DATA_BLOCK "DB_DP"   // DB85
{ S7_Optimized_Access := 'FALSE' }
// stored: AutoNumber false
   VAR RETAIN
      Anz_DP : Int := 2;   // * Anzahl Dosierpumpen
      Offset : Int := 20;   // * Beginn Daten
      leng_Pos : Int := 20;   // * Länge Daten
      DP_Nr : Int := 0;   // Nummer der aktuell bearbeiteten Pumpe
      Sekunden_Takt : Bool := FALSE;   // merkt sich den Sekundentakt
      Minuten_Takt : Bool := FALSE;   // eine Minute ist um (für einen Umlauf an)
      HandeventTakt : Bool := FALSE;   // zyklischer Abstand Meldung manuelle Zugabe
      res1 : Bool := FALSE;
      res2 : Bool := FALSE;
      res3 : Bool := FALSE;
      res4 : Bool := FALSE;
      res5 : Bool := FALSE;
      AM_Minute : Byte := 16#32;   // Altmerker Minute
      MinCount : Int := 1;   // Minutenzähler (10min)
      CheckPU : Int := 0;   // Kontrollpumpe
      resI : Int := 0;
      resD1 : DWord := 16#0000_0000;
      DP : Array[0..20] of Struct   // * Feldlänge anpassen
         Typ : Byte;   // *VAT 0=Menge Zeit,1=Menge Pulse,2=Handzugabe,5=H2O
         LaZa_Nr : Byte;   // *VAT Ladungszähler-Nr.
         EventTime : Int;   // 0=jede Dosierung sonst Zeit in Minuten
         Rest_EventTime : Int;   // Restzeit bis nächstes Event
         DP_Start : Bool;   // Start Dosierpumpe (auch extern 1 Autowert)
         DP_OFF : Bool;   // ext.Abschaltg. zB.Motorschutz oä.
         DP_Hand : Bool;   // Start eine Handzugabe
         DP_Strg : Bool;   // Störung Dosierpumpe
         DP_Imp : Bool;   // externer Zählimpuls
         DP_Niv : Bool;   // Niveau max erreicht
         DP_IN6 : Bool;
         DP_IN7 : Bool;
         DP_IN8 : Bool;
         Dosi_akt : Bool;   // Nachdosierung aktiv
         AM_Dosi : Bool;   // Altmerker Dosierung
         Meldung : Bool;   // Dosierung melden
         AM_Strg : Bool;   // Altmerker Störung
         DP_ext_Imp : Bool;   // Pumpe wird extern betrieben (Impuls wird als Eingang geliefert)
         res4 : Bool;
         AM_DP_Start : Bool;   // Merker DP Start
         RestZeit : Int;   // Restzeit Zähler Dosierimpuls/Pausenzeit
         DosMenge_Auto : Real;   // Dosiermenge Automatik
         DosMenge_Hand : Real;   // Dosiermenge Handzugabe
         ZeitBasis : Byte;   // Zeitbasis für Kalibrierung 0=s 1=min 2=h
         Korr_Einheit : Byte;   // ggf.Korrektur der Einheit
      END_STRUCT;
   END_VAR
BEGIN
   DP[0..20].Typ := 16#00;
   DP[0..20].LaZa_Nr := 16#00;
   DP[0..20].EventTime := 0;
   DP[0..7].Rest_EventTime := 1;
   DP[8..20].Rest_EventTime := 0;
   DP[0..20].DP_Start := FALSE;
   DP[0..20].DP_OFF := FALSE;
   DP[0..20].DP_Hand := FALSE;
   DP[0..20].DP_Strg := FALSE;
   DP[0..20].DP_Imp := FALSE;
   DP[0..20].DP_Niv := FALSE;
   DP[0..20].DP_IN6 := FALSE;
   DP[0..20].DP_IN7 := FALSE;
   DP[0..20].DP_IN8 := FALSE;
   DP[0..20].Dosi_akt := FALSE;
   DP[0..20].AM_Dosi := FALSE;
   DP[0..7].Meldung := TRUE;
   DP[8..20].Meldung := FALSE;
   DP[0..20].AM_Strg := FALSE;
   DP[0..20].DP_ext_Imp := FALSE;
   DP[0..20].res4 := FALSE;
   DP[0..20].AM_DP_Start := FALSE;
   DP[0..20].RestZeit := 0;
   DP[0..20].DosMenge_Auto := 0.0;
   DP[0..20].DosMenge_Hand := 0.0;
   DP[0..20].ZeitBasis := 16#00;
   DP[0..20].Korr_Einheit := 16#00;
END_DATA_BLOCK

DATA_BLOCK "DB_Dosi_Overview"   // DB88
{ S7_Optimized_Access := 'FALSE' }
// stored: AutoNumber false
   VAR RETAIN
      LZ_Count : Array[1..13] of DWord;   // * erst DZ je 1 DW
      DP_Count : Array[1..40] of DWord;   // * dann DP je 2 DW (Auto/Hand)(Feldlänge := DZ + 2*DP)
   END_VAR
BEGIN
   LZ_Count[1..13] := 16#0000_0000;
   DP_Count[1..40] := 16#0000_0000;
END_DATA_BLOCK

DATA_BLOCK "DB_NSP"   // DB96
{ S7_Optimized_Access := 'FALSE' }
// stored: AutoNumber false
   VAR RETAIN
      Anz_Per_Cyc : Int := 10;   // * Anzahl Positionen pro Zyklus (kleiner eine Sekunde müssen alle durch sein)
      Offset : Int := 20;   // Beginn Datenblock
      leng : Int := 20;   // Länge einer Struktue
      akt_NSP : Int := 55;   // aktueller Eintrag
      Test_on : Bool := TRUE;   // Testfunktion aktiv (nicht gewählte NSP/SPR aus)
      Test_akt : Bool := FALSE;   // Test Einzelpos (TestNr) aktiv
      Test_start : Bool := FALSE;   // Test angemeldet erster Umlauf alles aus
      Sekunde : Bool := FALSE;   // Sekunde M2.5 war ein
      Takt : Bool := FALSE;   // Takt (Sekunde) Zeiten zählen
      AMS_Reset : Bool := FALSE;   // Reset gefordert
      AMS_new : Bool := FALSE;   // Meldung neu schicken
      SammelWarn : Bool := FALSE;   // SammelWarnung min/max über alle Pos.
      Sammelstoer : Bool := FALSE;   // Sammelstörung Timeout über alle Pos.
      noMD_opt_max : Bool := FALSE;   // Überlauf nicht optisch melden
      noMD_opt_min : Bool := FALSE;   // Niveau min nicht optisch melden
      noMD_opt_Zeit : Bool := FALSE;   // Zeitüberschreit. nicht optisch melden
      noMD_aku_max : Bool := FALSE;   // Überlauf nicht akustisch melden
      noMD_aku_min : Bool := FALSE;   // Niveau min nicht akustisch melden
      noMD_aku_Zeit : Bool := FALSE;   // Zeitüberschreit. nicht akustisch melden
      Reset : Bool := FALSE;   // Reset Timeout NS
      TestNr : Int := 0;   // Nachspeisung für Test (alle anderen werden nicht bearbeitet)
      temp_Warn : Bool := FALSE;
      temp_STM : Bool := FALSE;
      resX122 : Bool := FALSE;
      resX123 : Bool := FALSE;
      resX124 : Bool := FALSE;
      resX125 : Bool := FALSE;
      resX126 : Bool := FALSE;
      resX127 : Bool := FALSE;
      resB1 : Byte := 16#00;
      resW1 : Int := 0;
      resD1 : DInt := 0;
      NSP : Array[1..30] of Struct
         NSP : Bool;   // Niveauregelung
         NST_in : Bool;   // Takt nach WT im Bad eingesetzt
         NST_out : Bool;   // Takt nach WT aus Bad ausgehoben
         SPR_in : Bool;   // Spritzen bei FW senkt
         SPR_out : Bool;   // Spritzen bei FW hebt
         SPR_expo : Bool;   // Spritzen während Expozeit
         SPR_Zeit : Bool;   // Spritzen feste Zeit nach Ausheben oder Einsetzen
         resTyp1 : Bool;   // ReserveTyp
         resTyp2 : Bool;   // ReserveTyp
         resTyp3 : Bool;   // ReserveTyp
         resTyp4 : Bool;   // ReserveTyp
         resTyp5 : Bool;   // ReserveTyp
         resTyp6 : Bool;   // ReserveTyp
         resTyp7 : Bool;   // ReserveTyp
         resTyp8 : Bool;   // ReserveTyp
         resTyp9 : Bool;   // ReserveTyp
         Freigabe : Bool;   // Freigabe Nachspeisung
         extern_Start : Bool;   // externe Aktivierung Taktung (zum Beispiel bei mehreren Pos)
         Niveau_ok : Bool;   // Niveau is ok Nachspeisung über Niveauregelung aus
         Nachspeisen : Bool;   // Nachspeisung aktiv --> Ventil auf / Pumpe an
         Spritzen : Bool;   // Spritzregister ein
         AL_Ueberlauf : Bool;   // Behälter Überlauf
         AL_Niv_min : Bool;   // Niveau zu niedrig --> Behälter leer
         AL_Zeit : Bool;   // Nachspeise-Zeitüberschreitung
         Restzeit_NSP : Int;   // Restzeit Nachspeisung
         TestNSP : Int;   // Testzeit Nachspeisung
         Restzeit_SPR : Int;   // Restzeit Spritzen
         VerzT : Int;   // Verzögerung Alarm Überlauf/Min-Niveau
         RestVerz : Int;   // Restzeit bis Alarm
         VerzNS_AL : Int;   // Verzögerung Alarm Nachspeisezeit zu gross
         RestNS_AL : Int;   // Restzeit bis Alarm
         AM_AL_min : Bool;   // Altmerker Alarm min
         AM_AL_Uel : Bool;   // Altmerker Alarm voll
         AM_AL_Zeit : Bool;   // Altmerker Alarm Nachspeise-Zeitüberschreitung
         AM_Bad_belegt : Bool;   // Altmerker Bad belegt
         AM_Reset : Bool;   // Altmerker RESET Nachspeise-Zeitüberschreitung
         res2 : Bool;
         res3 : Bool;
         res4 : Bool;
         SprFree : Bool;   // Spritzregister nicht bedienen (keine Ausgabe weder on noch off) Bedienung ext.
         NSPFree : Bool;   // Nachspeisung nicht bedienen (keine Ausgabe weder on noch off) Bedienung extern
         Warte_NSPT : Bool;   // getaktete Nachspeisung nicht abarbeiten
         res8 : Bool;
         res9 : Bool;
         res10 : Bool;
         res11 : Bool;
         res12 : Bool;
      END_STRUCT;
   END_VAR
BEGIN
   NSP[1..30].NSP := FALSE;
   NSP[1..30].NST_in := FALSE;
   NSP[1..30].NST_out := FALSE;
   NSP[1..30].SPR_in := FALSE;
   NSP[1..25].SPR_out := FALSE;
   NSP[26].SPR_out := TRUE;
   NSP[27..29].SPR_out := FALSE;
   NSP[30].SPR_out := TRUE;
   NSP[1..30].SPR_expo := FALSE;
   NSP[1..30].SPR_Zeit := FALSE;
   NSP[1..30].resTyp1 := FALSE;
   NSP[1..30].resTyp2 := FALSE;
   NSP[1..30].resTyp3 := FALSE;
   NSP[1..30].resTyp4 := FALSE;
   NSP[1..30].resTyp5 := FALSE;
   NSP[1..30].resTyp6 := FALSE;
   NSP[1..30].resTyp7 := FALSE;
   NSP[1..30].resTyp8 := FALSE;
   NSP[1..30].resTyp9 := FALSE;
   NSP[1..30].Freigabe := FALSE;
   NSP[1..30].extern_Start := FALSE;
   NSP[1..30].Niveau_ok := FALSE;
   NSP[1..30].Nachspeisen := FALSE;
   NSP[1..30].Spritzen := FALSE;
   NSP[1..30].AL_Ueberlauf := FALSE;
   NSP[1..30].AL_Niv_min := FALSE;
   NSP[1..30].AL_Zeit := FALSE;
   NSP[1..30].Restzeit_NSP := 0;
   NSP[1..30].TestNSP := 0;
   NSP[1..30].Restzeit_SPR := 0;
   NSP[1..30].VerzT := 0;
   NSP[1..30].RestVerz := 0;
   NSP[1..30].VerzNS_AL := 0;
   NSP[1..30].RestNS_AL := 0;
   NSP[1..30].AM_AL_min := FALSE;
   NSP[1..30].AM_AL_Uel := FALSE;
   NSP[1..30].AM_AL_Zeit := FALSE;
   NSP[1..30].AM_Bad_belegt := FALSE;
   NSP[1..30].AM_Reset := FALSE;
   NSP[1..30].res2 := FALSE;
   NSP[1..30].res3 := FALSE;
   NSP[1..30].res4 := FALSE;
   NSP[1..30].SprFree := FALSE;
   NSP[1..30].NSPFree := FALSE;
   NSP[1..30].Warte_NSPT := FALSE;
   NSP[1..30].res8 := FALSE;
   NSP[1..30].res9 := FALSE;
   NSP[1..30].res10 := FALSE;
   NSP[1..30].res11 := FALSE;
   NSP[1..30].res12 := FALSE;
END_DATA_BLOCK

DATA_BLOCK "DB_Panel_DP"   // DB86
{ S7_Optimized_Access := 'FALSE' }
AUTHOR : KHE_RE
NAME : DB_LADUN
VERSION : 2.0
// stored: AutoNumber false
   VAR RETAIN
      Anz_DP : Int := 8;   // * Anzahl Dosierpumpen
      Offset : Int := 20;   // * Beginn Daten
      Length : Int := 40;   // * Länge Daten
      res60 : Bool := FALSE;
      resB7 : Byte := 16#00;
      resB8 : Byte := 16#00;
      resB9 : Byte := 16#00;
      resB10 : Byte := 16#00;
      resB11 : Byte := 16#00;
      resD12 : DWord := 16#0000_0000;
      resD16 : DWord := 16#0000_0000;
      DoPu : Array[1..20] of Struct   // * Feldlänge anpassen
         Impulsdauer : Int;   // * Laufzeit Dosierimpuls [1/10 sec] (Falls keine Einstellmöglichkeit am PC)
         Impulspause : Int;   // * Pausenzeit zwischen zwei Impulsen [1/10 sec](Falls keine Einstellmöglichkeit
         resI : Int;
         Ein : Bool;   // Pumpe dauerhaft ein
         Auto : Bool;   // Pumpe Automatikbetrieb ein
         Kalibrierung : Bool;   // Pumpe in Kalibrierung
         res1 : Bool;
         res2 : Bool;
         Hand : Bool;   // Handdosierung läuft
         ON : Bool;   // DuPu läuft
         STM : Bool;   // DoPu Störung
         Kali_Start : Bool;   // Kalibrierung starten
         Kali_Stop : Bool;   // Kalibrierung anhalten
         res8 : Bool;
         res9 : Bool;
         res10 : Bool;
         res11 : Bool;
         res12 : Bool;
         res13 : Bool;
         Pumpleistung : Real;   // ml/s ml/Imp ....
         Zugabe_Hand : Real;   // ml
         Zugabe_Auto : Real;   // ml, ml/dm2
         RestDosierWert : Real;   // ml, Liter, g, kg usw.
         Kalibrierwert : Real;
         resD1 : DWord;
         resD2 : DWord;
         Kali_Count : DInt;   // Zählzelle Kalibrierdauer
      END_STRUCT;
   END_VAR
BEGIN
   DoPu[1..20].Impulsdauer := 1;
   DoPu[1..20].Impulspause := 1;
   DoPu[1..20].resI := 1;
   DoPu[1..20].Ein := FALSE;
   DoPu[1..4].Auto := TRUE;
   DoPu[5..20].Auto := FALSE;
   DoPu[1..20].Kalibrierung := FALSE;
   DoPu[1..20].res1 := FALSE;
   DoPu[1..20].res2 := FALSE;
   DoPu[1..20].Hand := FALSE;
   DoPu[1..20].ON := FALSE;
   DoPu[1..20].STM := FALSE;
   DoPu[1..20].Kali_Start := FALSE;
   DoPu[1..20].Kali_Stop := FALSE;
   DoPu[1..20].res8 := FALSE;
   DoPu[1..20].res9 := FALSE;
   DoPu[1..20].res10 := FALSE;
   DoPu[1..20].res11 := FALSE;
   DoPu[1..20].res12 := FALSE;
   DoPu[1..20].res13 := FALSE;
   DoPu[1..8].Pumpleistung := 0.1;
   DoPu[9..20].Pumpleistung := 0.0;
   DoPu[1..20].Zugabe_Hand := 0.0;
   DoPu[1..4].Zugabe_Auto := 10.0;
   DoPu[5..20].Zugabe_Auto := 0.0;
   DoPu[1].RestDosierWert := 0.0;
   DoPu[2].RestDosierWert := 0.09993901;
   DoPu[3..4].RestDosierWert := 0.09999623;
   DoPu[5..20].RestDosierWert := 0.0;
   DoPu[1..20].Kalibrierwert := 0.0;
   DoPu[1..20].resD1 := 16#0000_0000;
   DoPu[1..20].resD2 := 16#0000_0000;
   DoPu[1..20].Kali_Count := 0;
END_DATA_BLOCK

DATA_BLOCK "DB_Panel_LZ"   // DB81
{ S7_Optimized_Access := 'FALSE' }
AUTHOR : KHE_RE
NAME : DB_LADUN
VERSION : 2.0
// stored: AutoNumber false
   VAR RETAIN
      Anz : Int := 0;   // wird aus DB1 übernommen
      Offset : Int := 20;   // * Beginn Daten
      Length : Int := 36;   // * Länge Daten
      resB6 : Byte := 16#00;
      resB7 : Byte := 16#00;
      resD8 : DWord := 16#0000_0000;
      resD12 : DWord := 16#0000_0000;
      resD16 : DWord := 16#0000_0000;
      Becken : Array[1..20] of Struct   // * Feldlänge anpassen
         Dosi_Int : DInt;   // Abstand zw. 2 Dosierungen (Sollw.)
         Dosi_Zaehl : DInt;   // Ladung nach letzter Dosierung (Istw.)
         Rest_Zaehl1 : DInt;
         Ladu_Zaehl1 : DInt;   // kont. Ladungszähler 1 (Soll/Istw.)
         Ladu_Zaehl2 : DInt;   // kont. Ladungszähler 2 (Soll/Istw.)
         Ladu_Zaehl3 : DInt;   // kont. Ladungszähler 3 (Soll/Istw.)
         Ladu_Zaehl4 : DInt;   // kont. Ladungszähler 4 (Soll/Istw.)
         Ladu_Zaehl5 : DInt;   // kont. Ladungszähler 5 (Soll/Istw.)
         Ladu_Zaehl6 : DInt;   // kont. Ladungszähler 6 (Soll/Istw.)
      END_STRUCT;
   END_VAR
BEGIN
   Becken[1..20].Dosi_Int := 1000;
   Becken[1..20].Dosi_Zaehl := 0;
   Becken[1..20].Rest_Zaehl1 := 0;
   Becken[1..20].Ladu_Zaehl1 := 0;
   Becken[1..20].Ladu_Zaehl2 := 0;
   Becken[1..20].Ladu_Zaehl3 := 0;
   Becken[1..20].Ladu_Zaehl4 := 0;
   Becken[1..20].Ladu_Zaehl5 := 0;
   Becken[1..20].Ladu_Zaehl6 := 0;
END_DATA_BLOCK

DATA_BLOCK "DB_Panel_OVERVIEW"   // DB50
{ S7_Optimized_Access := 'FALSE' }
// stored: AutoNumber false
   VAR
      BA : Struct
         Not_Aus : Bool := FALSE;   // Not-Aus ist betätigt
         free0 : Bool := FALSE;   // sonst Anlage vom PC bedienen, nur bei BA-Schalter auf Auto
         free1 : Bool := FALSE;   // sonst Automatikbetrieb ist nicht freigegeben
         Tippbetrieb : Bool := FALSE;   // Tippbetrieb
         Handbetrieb : Bool := TRUE;   // Handbetrieb
         Automat_ein : Bool := FALSE;   // Automatikbetrieb möglich
         Automat_aus : Bool := FALSE;   // Automatikbetrieb nicht möglich
         Anlauf_Auto : Bool := FALSE;   // Anlauf Automatik für Scanvorgang WT-Positionen auf letzte Automatikposition
         Einfahr_Stop : Bool := FALSE;   // Stoppt die Einfahrt von WT in die Anlage(Feierabendprogramm)
         Mess_on : Bool := FALSE;   // Einmessung aktiv
         Taktwechsel : Bool := FALSE;   // Taktwechsel durchführen
         SIM_HISPEED : Bool := FALSE;   // Simulation erfolgt mit doppelter Geschwindigkeit
         Simulation : Bool := TRUE;   // Simulation eingeschaltet
         COM_RST : Bool := TRUE;   // Complete Restart
         FP_Automat_ein : Bool := FALSE;   // Flankenmerker positive Flanke Taste Automat ein
         newConfig : Bool := FALSE;   // neue Konfiguration (Daten neu verteilen)
      END_STRUCT;
      Offset : Int := 50;
      Leng : Int := 40;
      resW : Word := 16#0000;
      resDW2 : DWord := 16#0000_0000;
      resDW3 : DWord := 16#0000_0000;
      last_Takt : DInt := 0;
      Taktzeit : DInt := 0;   // Zeit die der Takt läuft
      Takt_Ware : DInt := 0;   // Zeit seit Ausfahrt letzte Fertigware
      resW1 : Word := 16#0000;
      Stop_Anlage : Byte := 16#00;   // ungleich 0-->Kettenbearbeitung anhalten
      Feierabend : Byte := 16#00;   // ungleich 0-->FEIERABENDPROGRAMM
      Sonder_BA : Byte := 16#00;   // ungleich 0-->ELEKTROLYSE, ENTMETALLISIEREN
      IST_Sonder_BA : Byte := 16#00;
      FB_FW_akt : Word := 16#0000;   // an Fernbedienung gewählter FW
      SPS_getaktet : Bool := TRUE;
      resDW9 : Word := 16#0000;
      Systime : DInt := 0;
      WT_Frueh : Byte := 16#00;   // Anzeige Anzahl der fertiggestellten WTs in der Frühschicht
      WT_Spaet : Byte := 16#15;   // Anzeige Anzahl der fertiggestellten WTs in der Spätschicht
      WT_Nacht : Byte := 16#00;   // Anzeige Anzahl der fertiggestellten WTs in der Nachtschicht
      resB : Byte := 16#00;
      resI : Int := 0;
      Pos : Array[1..30] of Struct   // * Feldlänge anpassen
         WT_Nr_lang : DInt;   // Warenträger-Nr lang
         WT_Nr_kurz : Byte;   // Warenträger-Nr kurz DB
         Stange_Nr : Byte;   // Warenstangen-Nr. (falls vorhanden)
         Soll_Expo : DInt;   // Sollwert Expositionszeit
         Rest_Expo : DInt;   // Verbleibende Expositionszeit
         BE_rdy : Bool;   // Beladestand bereit
         BE_leer : Bool;   // Beladestand leer
         BE_WT_vorhanden : Bool;   // Beladestand mit nicht aufgebbaren WT belegt
         BE_verriegelt : Bool;   // Beladestand angedockt und verriegelt(arretiert)
         BE_gelb : Bool;
         BE_rot : Bool;
         BE_Charge_ok : Bool;   // Behandlung fehlerfrei
         BE_Charge_nok : Bool;   // Fehler bei Behandlung
         Sonderfkt : Byte;   // Sonderfunktionen frei verwendbar(WT-Kennung)
         priorisiert : Bool;   // priorisierter WT im Bad
         in_Anlage : Bool;   // will in die Anlage
         in_Entm : Bool;   // will in die Entmetallisierung
         aus_Anlage : Bool;   // kommt aus der Anlage
         aus_Entm : Bool;   // kommt aus der Entmetallisierung
         Speicher : Bool;   // Speicherprogramm
         Warnung : Bool;   // in Position wurde eine Warnung ausgelöst
         Alarm : Bool;   // in position wurde ein Alarm ausgelöst
         belegt : Bool;   // Bad belegt
         Trommel : Bool;   // Trommelware im Bad
         Leer_WT : Bool;   // Leerstange im Bad
         Vorruf : Bool;   // Vorruf für Fahrwagen ausgelößt
         fertig : Bool;   // Expozeit abgelaufen WT zu Abholung bereit
         Sperre_in : Bool;   // Einfahrsperre
         Sperre_FW : Bool;   // Überfahrsperre
         Sperre_out : Bool;   // Ausfahrsperre
         Befx : Int;   // Befehlsindex
         Vorsperre : Bool;   // Einfahrsperre angemeldet
         Dummy1 : Bool;   // Dummy auf Dummyposition abgelegt
         Dummy2 : Bool;   // Dummy auf Mittenposition abgelegt
         Dkl_auf_Pos : Bool;   // Deckel auf dieser Position
         Expo_Warn : Bool;   // Warnung: Toleranzüberschreitg.Expozeit
         Expo_Off : Bool;   // Expositionszeit eingefroren
         NSP_ON : Bool;   // Laufanzeige Nachspeisung
         SPR_ON : Bool;   // Laufanzeige Spritzregister
         WT_Typ : Byte;   // Art des Warenträgers (z.Bsp. bei fester Zuordnung Ware-WT)
         Verweilzeit : DInt;   // Verweilzeit in s
         Sonderwert_1 : Real;   // z.B. Gewicht bei Beladestand
         Fertigzeitpunkt : DInt;   // Systemzeit PC, wann WT voraussichtlich fertig
         Sonderwert_2 : Real;   // z.B. Gewicht bei Beladestand
         resb : Byte;
         Dkl_zu : Bool;   // Deckel ist zu
         Dkl_auf : Bool;   // Deckel ist auf
         res392 : Bool;
         res393 : Bool;
         PendelHub : Bool;   // Mehrfachtauchen
         res395 : Bool;
         res396 : Bool;
         res397 : Bool;
      END_STRUCT;
   END_VAR
BEGIN
   Pos[1..30].WT_Nr_lang := 0;
   Pos[1..30].WT_Nr_kurz := 16#00;
   Pos[1..30].Stange_Nr := 16#00;
   Pos[1].Soll_Expo := 0;
   Pos[2].Soll_Expo := 360;
   Pos[3].Soll_Expo := 60;
   Pos[4..7].Soll_Expo := 1260;
   Pos[8..9].Soll_Expo := 90;
   Pos[10].Soll_Expo := 75;
   Pos[11..12].Soll_Expo := 5;
   Pos[13..14].Soll_Expo := 75;
   Pos[15..16].Soll_Expo := 5;
   Pos[17].Soll_Expo := 75;
   Pos[18].Soll_Expo := 5;
   Pos[19].Soll_Expo := 75;
   Pos[20].Soll_Expo := 5;
   Pos[21].Soll_Expo := 10;
   Pos[22].Soll_Expo := 360;
   Pos[23..27].Soll_Expo := 5;
   Pos[28].Soll_Expo := 0;
   Pos[29..30].Soll_Expo := 5;
   Pos[1..30].Rest_Expo := 0;
   Pos[1].BE_rdy := TRUE;
   Pos[2..30].BE_rdy := FALSE;
   Pos[1..30].BE_leer := FALSE;
   Pos[1..30].BE_WT_vorhanden := FALSE;
   Pos[1].BE_verriegelt := TRUE;
   Pos[2..30].BE_verriegelt := FALSE;
   Pos[1..30].BE_gelb := FALSE;
   Pos[1..30].BE_rot := FALSE;
   Pos[1..30].BE_Charge_ok := FALSE;
   Pos[1..30].BE_Charge_nok := FALSE;
   Pos[1..30].Sonderfkt := 16#00;
   Pos[1..30].priorisiert := FALSE;
   Pos[1..30].in_Anlage := FALSE;
   Pos[1..30].in_Entm := FALSE;
   Pos[1..30].aus_Anlage := FALSE;
   Pos[1..30].aus_Entm := FALSE;
   Pos[1..30].Speicher := FALSE;
   Pos[1..30].Warnung := FALSE;
   Pos[1..30].Alarm := FALSE;
   Pos[1..30].belegt := FALSE;
   Pos[1..30].Trommel := FALSE;
   Pos[1..30].Leer_WT := FALSE;
   Pos[1..30].Vorruf := FALSE;
   Pos[1..30].fertig := FALSE;
   Pos[1..30].Sperre_in := FALSE;
   Pos[1..30].Sperre_FW := FALSE;
   Pos[1..30].Sperre_out := FALSE;
   Pos[1..30].Befx := 0;
   Pos[1..30].Vorsperre := FALSE;
   Pos[1..30].Dummy1 := FALSE;
   Pos[1..30].Dummy2 := FALSE;
   Pos[1..30].Dkl_auf_Pos := FALSE;
   Pos[1..30].Expo_Warn := FALSE;
   Pos[1..30].Expo_Off := FALSE;
   Pos[1..30].NSP_ON := FALSE;
   Pos[1..30].SPR_ON := FALSE;
   Pos[1..30].WT_Typ := 16#00;
   Pos[1..30].Sonderwert_1 := 0.0;
   Pos[1..30].Fertigzeitpunkt := 0;
   Pos[1..30].Sonderwert_2 := 0.0;
   Pos[1..30].resb := 16#00;
   Pos[1..30].Dkl_zu := FALSE;
   Pos[1..30].Dkl_auf := FALSE;
   Pos[1..30].res392 := FALSE;
   Pos[1..30].res393 := FALSE;
   Pos[1..30].PendelHub := FALSE;
   Pos[1..30].res395 := FALSE;
   Pos[1..30].res396 := FALSE;
   Pos[1..30].res397 := FALSE;
END_DATA_BLOCK

DATA_BLOCK "DB_Zaehler"   // DB80
{ S7_Optimized_Access := 'FALSE' }
AUTHOR : KHE_RE
NAME : DB_LADUN
VERSION : 2.0
// stored: AutoNumber false
   VAR RETAIN
      Anz_Beck : Int := 2;   // wird aus DB1 übernommen
      Offset : Int := 40;   // * Beginn Daten
      leng_Pos : Int := 40;   // * Länge Daten
      Tag_neu : Bool := FALSE;
      Wo_neu : Bool := FALSE;
      Mo_neu : Bool := FALSE;
      res3 : Bool := FALSE;
      res4 : Bool := FALSE;
      res5 : Bool := FALSE;
      res6 : Bool := FALSE;
      AM_Takt : Bool := FALSE;
      I_Time : Byte := 16#01;
      Beck_Nr : Byte := 16#02;
      resb0 : Byte := 16#00;
      MZ_T : Byte := 16#10;   // Merkzelle akt.Tag
      MZ_W : Byte := 16#00;   // Merkzelle akt.Woche
      MZ_M : Byte := 16#06;   // Merkzelle akt.Monat
      Beck_ext : Byte := 16#00;   // Becken-Nr. für externe Dosierzähler
      Wert_Ext : Real := 0.0;   // ext. Zählwert (siehe FC6)
      resDW2 : DWord := 16#0000_0000;
      resDW3 : DWord := 16#0000_0000;
      resDW4 : DWord := 16#0000_0000;
      DosMenge_Typ7 : DWord := 16#0000_0000;
      resDW5 : DWord := 16#0000_0000;
      resW : Word := 16#0000;
      Becken : Array[1..20] of Struct   // * Feldlänge anpassen
         Typ : Byte;   // Typ 0=Ah, 1=Amin, 4=dm2, 6=ext.Zähler(FC6) 8=ext.Ah-Zähler
         Anz_Bad : Byte;   // Anz. des Bäder im Becken
         Input : Array[1..10] of Struct   // Liste der Bäder
            Pos : Int;
         END_STRUCT;
         Zaehl_int : Real;   // interner Restzähler
         Dig_Inp : Byte;   // Dig. Eing. (res.)
         Event : Bool;   // Event Mengenlimit erreicht
         Stop : Bool;   // Dosierzähler gestoppt (von DoPu o.ä.)
         res2 : Bool;
         res3 : Bool;
         res4 : Bool;
         res5 : Bool;
         res6 : Bool;
         Anf_Stp : Bool;   // kumulat.Anforderung Stop DoZa
         resW : Word;
         EventCount : Real;   // Zählzelle für Events
         ext_Val : Real;   // externer Zählwert
         AM_belegt : Word;   // Altmerker Pos.belegt
      END_STRUCT;
   END_VAR
BEGIN
   Becken[1..2].Typ := 16#05;
   Becken[3..20].Typ := 16#00;
   Becken[1..2].Anz_Bad := 16#06;
   Becken[3..20].Anz_Bad := 16#00;
   Becken[1].Input[1].Pos := 1;
   Becken[1].Input[2].Pos := 2;
   Becken[1].Input[3].Pos := 3;
   Becken[1].Input[4].Pos := 4;
   Becken[1].Input[5].Pos := 5;
   Becken[1].Input[6].Pos := 6;
   Becken[1].Input[7..10].Pos := 0;
   Becken[2].Input[1].Pos := 13;
   Becken[2].Input[2].Pos := 14;
   Becken[2].Input[3].Pos := 15;
   Becken[2].Input[4].Pos := 16;
   Becken[2].Input[5].Pos := 17;
   Becken[2].Input[6].Pos := 18;
   Becken[2].Input[7..10].Pos := 0;
   Becken[3].Input[1..10].Pos := 0;
   Becken[4].Input[1..10].Pos := 0;
   Becken[5].Input[1..10].Pos := 0;
   Becken[6].Input[1..10].Pos := 0;
   Becken[7].Input[1..10].Pos := 0;
   Becken[8].Input[1..10].Pos := 0;
   Becken[9].Input[1..10].Pos := 0;
   Becken[10].Input[1..10].Pos := 0;
   Becken[11].Input[1..10].Pos := 0;
   Becken[12].Input[1..10].Pos := 0;
   Becken[13].Input[1..10].Pos := 0;
   Becken[14].Input[1..10].Pos := 0;
   Becken[15].Input[1..10].Pos := 0;
   Becken[16].Input[1..10].Pos := 0;
   Becken[17].Input[1..10].Pos := 0;
   Becken[18].Input[1..10].Pos := 0;
   Becken[19].Input[1..10].Pos := 0;
   Becken[20].Input[1..10].Pos := 0;
   Becken[1..20].Zaehl_int := 0.0;
   Becken[1..20].Dig_Inp := 16#00;
   Becken[1..20].Event := FALSE;
   Becken[1..20].Stop := FALSE;
   Becken[1..20].res2 := FALSE;
   Becken[1..20].res3 := FALSE;
   Becken[1..20].res4 := FALSE;
   Becken[1..20].res5 := FALSE;
   Becken[1..20].res6 := FALSE;
   Becken[1..20].Anf_Stp := FALSE;
   Becken[1..20].resW := 16#0000;
   Becken[1..20].EventCount := 0.0;
   Becken[1..20].ext_Val := 0.0;
   Becken[1..20].AM_belegt := 16#0000;
END_DATA_BLOCK

DATA_BLOCK "DB_BE_Stand"   // DB4
{ S7_Optimized_Access := 'FALSE' }
// stored: AutoNumber false
   VAR RETAIN
      Anzahl : Int := 6;   // * Anzahl der BE-/Entladestände
      leng : Int := 12;   // * Länge einer Struktur
      Offset : Int := 10;   // * Beginn des Datenfeldes
      Next : Byte := 16#00;   // nächster Wt für die Anlage
      Entm : Byte := 16#00;   // nächster Wt für die Entmetallisierung
      AnfQ : Byte := 16#00;   // Anforderung Quelle
      AnfZ : Byte := 16#00;   // Anforderung Ziel
      Stand : Array[1..6] of Struct   // * Feldlänge anpassen
         Pos_Nr : USInt;
         Aufgabe_erlaubt : Bool;   // Aufgabe ist möglich
         kein_WT : Bool;   // Stand ist leer (WT ist weder physikalisch noch logisch vorhanden)
         WT_aufgegeben : Bool;   // Warenträger ist aufgegeben
         verriegelt : Bool;   // Bedienung durch FW möglich
         gelb : Bool;
         rot : Bool;
         Charge_ok : Bool;   // Behandlung war fehlerfrei
         Charge_nok : Bool;   // Behandlung war gestört
         IN_innen : Bool;   // Wagen angedockt
         IN_aussen : Bool;   // Wagen im Beladebereich
         IN_Belegt : Bool;   // WT auf Wagen
         IN_Freigabe : Bool;   // Freigabetaste (wennvorhanden über Flankenmerker Bit4.0)
         OUT_Sperre_in : Bool;   // Einfahrsperre
         OUT_Sperre_FW : Bool;   // Überfahrsperre
         OUT_Sperre_out : Bool;   // Ausfahrsperre
         OUT_FW_kommt : Bool;   // Meldung FW kommt
         Del_Count : Byte;   // Sekundenzähler zum löschen der WT-Info
         AM_Freigabe : Bool;   // Altmerker Freigabetaste
         AM_Wagen : Bool;   // Altmerker Wagen vorhanden
         res3 : Bool;
         Trommel_BE : Bool;   // Trommelstand
         Gestell_BE : Bool;   // Gestellstand
         Ausf_Ware : Bool;   // Ausfahrt Ware erlaubt
         Ausf_Entm : Bool;   // Ausfahrt entmetallisierte Gestelle
         last_WT_Trommel : Bool;   // letzter WT war / ist Trommel
         Anf_Pos : Byte;   // Position die BE-Anfordert
         last_WT : DInt;   // letzte WT-Nr-lang
         Del_All : Bool;   // 0=Programm löschen 1=gesamten WT löschen
         Auto_Delete : Bool;   // automatisches löschen fertiger WT
         Afg_WT_Nr : Bool;   // Aufgabe auch bei WT_Nr_lang<>0 erlaubt
         res1 : Bool;
         res2 : Bool;
         res4 : Bool;
         res5 : Bool;
         schnell : Bool;
         resB : Byte;
      END_STRUCT;
      Langware_vorn : Bool;
      Langware_hinten : Bool;
   END_VAR
BEGIN
   Stand[1].Pos_Nr := 25;
   Stand[2].Pos_Nr := 26;
   Stand[3].Pos_Nr := 27;
   Stand[4].Pos_Nr := 28;
   Stand[5].Pos_Nr := 29;
   Stand[6].Pos_Nr := 30;
   Stand[1..5].Aufgabe_erlaubt := FALSE;
   Stand[1..3].kein_WT := TRUE;
   Stand[4..5].kein_WT := FALSE;
   Stand[1..5].WT_aufgegeben := FALSE;
   Stand[1].verriegelt := FALSE;
   Stand[2].verriegelt := TRUE;
   Stand[3..5].verriegelt := FALSE;
   Stand[1..5].gelb := FALSE;
   Stand[1..5].rot := FALSE;
   Stand[1..5].Charge_ok := FALSE;
   Stand[1..5].Charge_nok := FALSE;
   Stand[1].IN_innen := FALSE;
   Stand[2].IN_innen := TRUE;
   Stand[3..5].IN_innen := FALSE;
   Stand[1].IN_aussen := FALSE;
   Stand[2].IN_aussen := TRUE;
   Stand[3..5].IN_aussen := FALSE;
   Stand[1..5].IN_Belegt := FALSE;
   Stand[1].IN_Freigabe := FALSE;
   Stand[2].IN_Freigabe := TRUE;
   Stand[3..5].IN_Freigabe := FALSE;
   Stand[1].OUT_Sperre_in := TRUE;
   Stand[2..5].OUT_Sperre_in := FALSE;
   Stand[1..5].OUT_Sperre_FW := FALSE;
   Stand[1..2].OUT_Sperre_out := TRUE;
   Stand[3..5].OUT_Sperre_out := FALSE;
   Stand[1..5].OUT_FW_kommt := FALSE;
   Stand[1].Del_Count := 16#05;
   Stand[2].Del_Count := 16#1E;
   Stand[3..5].Del_Count := 16#00;
   Stand[1..5].AM_Freigabe := FALSE;
   Stand[1..2].AM_Wagen := TRUE;
   Stand[3..5].AM_Wagen := FALSE;
   Stand[1..5].res3 := FALSE;
   Stand[1..5].Trommel_BE := FALSE;
   Stand[1..5].Gestell_BE := FALSE;
   Stand[1..5].Ausf_Ware := FALSE;
   Stand[1..5].Ausf_Entm := FALSE;
   Stand[1..5].last_WT_Trommel := FALSE;
   Stand[1..5].Anf_Pos := 16#00;
   Stand[1..5].last_WT := 0;
   Stand[1..2].Del_All := TRUE;
   Stand[3..5].Del_All := FALSE;
   Stand[1].Auto_Delete := FALSE;
   Stand[2].Auto_Delete := TRUE;
   Stand[3..5].Auto_Delete := FALSE;
   Stand[1..5].Afg_WT_Nr := FALSE;
   Stand[1..5].res1 := FALSE;
   Stand[1..5].res2 := FALSE;
   Stand[1..5].res4 := FALSE;
   Stand[1..5].res5 := FALSE;
   Stand[1..5].schnell := FALSE;
   Stand[1..5].resB := 16#00;
END_DATA_BLOCK

DATA_BLOCK "DB_Prog_edit"   // DB800
{ S7_Optimized_Access := 'FALSE' }
// stored: AutoNumber false
   VAR RETAIN
      akt_edit_prog : Int;
      akt_Aufgabe_Prog : Int;
      old_Aufgabe_Prog : Int;   // Hilfsvariable um Programm in Aufgabestruktur zu kopieren
      resW : Int;
      resW_1 : Int;
      resD : DInt;
      Variante : USInt;   // 1=KSvl, 2=KSvr, 3=GOli, 4= GOre,5=KShl, 6=kshr, 7=LSv(BE1), 8= LSh(BE5)
      StandNr : USInt;
      GZ_Charge : DInt;
      Prog : Array[1..100] of Struct
         "Name" : String[100];
         Geometrie : USInt;   // 0=k.A., 1=KS, 2=LS, 3=GO
         ParaByte : USInt;   // .0=lgsm senken, .1=lgsm heben
         Faktor_ATZ : Real;
         resD : DInt;
         resW : Int;
         CM03_VorSpuel : Struct
            Expo : Time_Of_Day;
            Anfahren : Bool;
            res : Bool;
            res_1 : Bool;
            res_2 : Bool;
            res_3 : Bool;
            res_4 : Bool;
            res_5 : Bool;
            res_6 : Bool;
            resB : Byte;
            resW : Int;
            resD : DInt;
         END_STRUCT;
         CM01_VorAetz : Struct
            Expo : Time_Of_Day;
            Anfahren : Bool;
            res : Bool;
            res_1 : Bool;
            res_2 : Bool;
            res_3 : Bool;
            res_4 : Bool;
            res_5 : Bool;
            res_6 : Bool;
            Anzahl_Voraetz : Byte;
            resW : Int;
            resD : DInt;
         END_STRUCT;
         CM03_SpuelVorAetz : Struct
            Expo : Time_Of_Day;
            Anfahren : Bool;
            res : Bool;
            res_1 : Bool;
            res_2 : Bool;
            res_3 : Bool;
            res_4 : Bool;
            res_5 : Bool;
            res_6 : Bool;
            resB : Byte;
            resW : Int;
            resD : DInt;
         END_STRUCT;
         CM01_Aetzen : Struct
            Expo : Time_Of_Day;
            resD : DInt;
            resD_1 : DInt;
         END_STRUCT;
         CM03_Spl_1 : Struct
            Expo : Time_Of_Day;
            resD : DInt;
            resD_1 : DInt;
         END_STRUCT;
         CM04_Spl_2 : Struct
            Expo : Time_Of_Day;
            resD : DInt;
            resD_1 : DInt;
         END_STRUCT;
      END_STRUCT;
      Prog_Aufgabe : Struct
         Prog : Struct
            "Name" : String[100];
            Geometrie : USInt;   // 0=k.A., 1=KS, 2=LS, 3=GO
            ParaByte : USInt;   // .0=lgsm senken, .1=lgsm heben
            Faktor_ATZ : Real;
            resD : DInt;
            resW : Int;
            CM03_VorSpuel : Struct
               Expo : Time_Of_Day;
               Anfahren : Bool;
               res : Bool;
               res_1 : Bool;
               res_2 : Bool;
               res_3 : Bool;
               res_4 : Bool;
               res_5 : Bool;
               res_6 : Bool;
               resB : Byte;
               resW : Int;
               resD : DInt;
            END_STRUCT;
            CM01_VorAetz : Struct
               Expo : Time_Of_Day;
               Anfahren : Bool;
               res : Bool;
               res_1 : Bool;
               res_2 : Bool;
               res_3 : Bool;
               res_4 : Bool;
               res_5 : Bool;
               res_6 : Bool;
               Anzahl_Voraetz : Byte;
               resW : Int;
               resD : DInt;
            END_STRUCT;
            CM03_SpuelVorAetz : Struct
               Expo : Time_Of_Day;
               Anfahren : Bool;
               res : Bool;
               res_1 : Bool;
               res_2 : Bool;
               res_3 : Bool;
               res_4 : Bool;
               res_5 : Bool;
               res_6 : Bool;
               resB : Byte;
               resW : Int;
               resD : DInt;
            END_STRUCT;
            CM01_Aetzen : Struct
               Expo : Time_Of_Day;
               resD : DInt;
               resD_1 : DInt;
            END_STRUCT;
            CM03_Spl_1 : Struct
               Expo : Time_Of_Day;
               resD : DInt;
               resD_1 : DInt;
            END_STRUCT;
            CM04_Spl_2 : Struct
               Expo : Time_Of_Day;
               resD : DInt;
               resD_1 : DInt;
            END_STRUCT;
         END_STRUCT;
         Korb_Nr : Int;
      END_STRUCT;
   END_VAR
BEGIN
END_DATA_BLOCK

DATA_BLOCK "DB_Techno"   // DB45
{ S7_Optimized_Access := 'FALSE' }
AUTHOR : RE
// stored: AutoNumber false
   VAR RETAIN
      DATEN_gueltig : Bool := FALSE;   // bit 0.0 rest vom Byte reserviert set:PC reset:SPS
      WT_NR_lng : DInt := 0;   // Warenträgernummer lang
      WT_NR_kurz : Byte := 16#00;   // wenn 0, dann Neuaufgabe eines WT
      STAND_NR : Byte := 16#00;   // wenn 0, dann Technologieänderung
      Oberflaeche : Real := 1.0;
      Prioritaet : Byte := 16#00;   // priorisierter WT Bit 12.0==1
      res : Bool := FALSE;
      res1 : Bool := FALSE;
      res2 : Bool := FALSE;
      res3 : Bool := FALSE;
      res4 : Bool := FALSE;
      res5 : Bool := FALSE;
      res6 : Bool := FALSE;
      res7 : Bool := FALSE;
      Korb_Nr : USInt;   // Korbnummer (fest)
      resByte : USInt;   // aktuelle Position
      Technologie : Int := 0;   // Technologie Code
      resW1 : Int := 0;
      resW2 : Int := 0;
      ParaByte : Byte := 16#00;   // Parameterbyte (inf. langsam Heben 22.1/Senken 22.0)
      WT_Typ : Byte := 16#00;   // Warenträgertyp B#16#11=KS, 12=LS, B#16#2x=GO
      resW3 : Int := 0;
      resD : DInt := 0;
      resD1 : DInt := 0;
      resD2 : DInt := 0;
      KorrPend : Real := 0.0;
      KorrATZ : Real := 0.0;
      Beginn_Daten : Int := 78;   // * Beginn des Technologiedatenblocks
      Ende_Daten : Int := 440;   // * Ende des Technologiedatenblocks
      resDW : DInt := 0;
      resDW1 : DInt := 0;
      resW4 : Int := 0;
      resW6 : Int := 0;
      AnzPendHub : Byte := 16#00;   // Anzahl Mehrfachhub
      WT_Kennung : Byte := 16#00;
      Speed_Up : Int := 0;   // Geschwindigkeitsbegrenzung Heben
      Speed_Dn : Int := 0;   // Geschwindigkeitsbegrenzung Senken
      Speed_Fahrt : Int := 0;   // Geschwindigkeitsbegrenzung Fahren (Ware)
      resI1 : Int := 0;
      resI2 : Int := 0;
      resI3 : Int := 0;
      resI4 : Int := 0;
      "Name" : String[100];
      stBefehle : Array[1..20] of Struct   // * bei Änderung anpassen
         Kennung : Byte;   // Befehlskennung
         FirstPos1 : Byte;   // erste Position, die angefahren werden kann
         Grpleng1 : Byte;   // Gruppenbad Länge
         FirstPos2 : Byte;
         Grpleng2 : Byte;
         Merker : Byte;
         Param_Ptr : Int;   // Pointer für Parameter
      END_STRUCT;
      stParam_Bereich : Array[1..100] of Byte;   // * bei Änderung oder Adressverschiebung anpassen
   END_VAR
BEGIN
   stBefehle[1..10].Kennung := 16#00;
   stBefehle[1..10].FirstPos1 := 16#00;
   stBefehle[1..10].Grpleng1 := 16#00;
   stBefehle[1..10].FirstPos2 := 16#00;
   stBefehle[1..10].Grpleng2 := 16#00;
   stBefehle[1..10].Merker := 16#00;
   stBefehle[1..10].Param_Ptr := 0;
   stParam_Bereich[1..100] := 16#00;
END_DATA_BLOCK

DATA_BLOCK "DB_WT1"   // DB101
{ S7_Optimized_Access := 'FALSE' }
AUTHOR : MS
// stored: AutoNumber false
   VAR RETAIN
      ANZAHL : Int := 10;   // * max. Anzahl der Befehle DB45 beachten!!
      OFFSET : Int := 180;   // * Beginn der Befehlskette
      LENG : Int := 8;   // * Befehlslänge in Byte
      WT_NR_lang : DInt;   // Warenträger-Nr. lang
      Oberflaeche : Real;   // Oberfläche in dm²
      Korb_Nr : USInt;   // Korbnummer (fest)
      POS : USInt;   // aktuelle Position
      Technologie : Int;   // Technologie Code
      priorisiert : Bool;   // WT ist proorisiert
      in_Anlage : Bool;   // will in die Anlage
      in_Entm : Bool;   // will in die Entmetallisierung
      aus_Anlage : Bool;   // kommt aus der Anlage
      aus_Entm : Bool;   // kommt aus der Entmetallisierung
      Speicher : Bool;   // Speicherprogramm
      FW_Pos : Bool;   // WT befindet sich am FW
      QT_Pos : Bool;   // WT befindet sich im QT
      Auto_Pos : USInt;   // Position für Automatikbetrieb
      Trommel : Bool;   // WT ist eine Trommel
      UT_Anforderung : Bool;   // Trockneranforderung erzeugt aus Befehl"FF"
      Stop : Bool;   // Stopbefehl aktiv
      Nassware : Bool;   // Nassware-Trichter am Entladestand anfordern
      TW_Pos : Bool;   // Warenträger ist noch in seiner Taktwechselposition
      noKorrBefx : Bool;   // Befehlsindex nicht korregieren
      noOPT_WT : Bool;   // kann nicht wie berechnet eingefahren werden
      last_Auto : Bool;   // letzter Umsetzvorgang erfolgte in Automatik
      Ziel_Pos_WT : USInt;   // Zielposition des WT für Korrektur beim Einsetzen
      lngsm_senken : Bool;   // langsam Senken
      lngsm_heben : Bool;   // langsam Heben
      lngsm_Fahrt : Bool;   // langsam Fahren
      WT_nok : Bool;   // Behandlungsfehler
      WT_151 : Bool;
      WT_161 : Bool;
      res226 : Bool;
      res227 : Bool;
      Alt_Befx : USInt;   // Befehlsindex in letzter Automatikposition
      Alt_Bereichstakte : USInt;   // Bereichstakte der letzten Automatikposition
      Alt_TW_Pos : USInt;
      Alt_Verweil : DInt;   // Verweilzeit der letzten Automatikposition
      Fertigzeitpunkt : DInt;   // Systemzeit PC, wann WT voraussichtlich fertig
      Meld_Pos : USInt;   // gemerkte Kollisionposition
      WT_Typ : Byte;   // Warenträgertyp (für die Zuordnung bestimmter Ware)
      End_Ziel_Pos : USInt;   // Zielposition an die der WT
      End_Ziel_QT_Pos : USInt;   // Position die ein verwendeter QT anfahren muß
      KorrPend : Real;   // Korrekturfaktor Pendelzeit
      KorrATZ : Real;   // Korrekturfaktor Abtropfzeit
      P_PNTER : Int;   // Parameter-Pointer
      B_PNTER : Int;   // Befehls-pointer
      SaveExpo : DInt;   // gerettete Expozeit bei Zwangsräumung
      Bereichstakte : USInt;   // Takt die der WT noch im aktuellen Behandlungsbereich verbringen muß
      Variante1 : Byte;
      Variante2 : Byte;
      Variante3 : Byte;
      Variante4 : Byte;
      Variante5 : Byte;
      akt_Ziel : Int;   // aktuelles Ziel aus FB9(FC120)
      akt_CMD : Byte;   // aktueller Befehl
      WT_Kennung : Byte;   // farbliche Markierung für PC
      Speed_Up : Int;
      Speed_Dn : Int;
      Speed_Fahrt : Int;
      resI : Int;
      Aufgabezeitpunkt : DInt;   // Systemzeit PC, wann WT aufgegeben wurde
      RestTakte : Int;   // Resttakte durch die Anlage
      "Name" : String[100];
      Befehl : Array[1..20] of Struct   // * Feldlänge anpassen DB45 beachten!!
         Kennung : Byte;   // Befehlskennung
         Startpos : Byte;   // Position
         Laenge : Byte;   // Länge
         Startpos2 : Byte;
         Laenge2 : Byte;
         Sonderparam : Byte;
         Param_Ptr : Int;   // Pointer für Parameter
      END_STRUCT;
      Param_Bereich : Array[1..100] of Byte;   // * Feldlänge anpassen DB45 beachten!!
   END_VAR
BEGIN
END_DATA_BLOCK

DATA_BLOCK "DB_WT10"   // DB110
{ S7_Optimized_Access := 'FALSE' }
AUTHOR : MS
// stored: AutoNumber false
   VAR RETAIN
      ANZAHL : Int := 10;   // * max. Anzahl der Befehle DB45 beachten!!
      OFFSET : Int := 180;   // * Beginn der Befehlskette
      LENG : Int := 8;   // * Befehlslänge in Byte
      WT_NR_lang : DInt;   // Warenträger-Nr. lang
      Oberflaeche : Real;   // Oberfläche in dm²
      Korb_Nr : USInt;   // Korbnummer (fest)
      POS : USInt;   // aktuelle Position
      Technologie : Int;   // Technologie Code
      priorisiert : Bool;   // WT ist proorisiert
      in_Anlage : Bool;   // will in die Anlage
      in_Entm : Bool;   // will in die Entmetallisierung
      aus_Anlage : Bool;   // kommt aus der Anlage
      aus_Entm : Bool;   // kommt aus der Entmetallisierung
      Speicher : Bool;   // Speicherprogramm
      FW_Pos : Bool;   // WT befindet sich am FW
      QT_Pos : Bool;   // WT befindet sich im QT
      Auto_Pos : USInt;   // Position für Automatikbetrieb
      Trommel : Bool;   // WT ist eine Trommel
      UT_Anforderung : Bool;   // Trockneranforderung erzeugt aus Befehl"FF"
      Stop : Bool;   // Stopbefehl aktiv
      Nassware : Bool;   // Nassware-Trichter am Entladestand anfordern
      TW_Pos : Bool;   // Warenträger ist noch in seiner Taktwechselposition
      noKorrBefx : Bool;   // Befehlsindex nicht korregieren
      noOPT_WT : Bool;   // kann nicht wie berechnet eingefahren werden
      last_Auto : Bool;   // letzter Umsetzvorgang erfolgte in Automatik
      Ziel_Pos_WT : USInt;   // Zielposition des WT für Korrektur beim Einsetzen
      lngsm_senken : Bool;   // langsam Senken
      lngsm_heben : Bool;   // langsam Heben
      lngsm_Fahrt : Bool;   // langsam Fahren
      WT_nok : Bool;   // Behandlungsfehler
      WT_151 : Bool;
      WT_161 : Bool;
      res226 : Bool;
      res227 : Bool;
      Alt_Befx : USInt;   // Befehlsindex in letzter Automatikposition
      Alt_Bereichstakte : USInt;   // Bereichstakte der letzten Automatikposition
      Alt_TW_Pos : USInt;
      Alt_Verweil : DInt;   // Verweilzeit der letzten Automatikposition
      Fertigzeitpunkt : DInt;   // Systemzeit PC, wann WT voraussichtlich fertig
      Meld_Pos : USInt;   // gemerkte Kollisionposition
      WT_Typ : Byte;   // Warenträgertyp (für die Zuordnung bestimmter Ware)
      End_Ziel_Pos : USInt;   // Zielposition an die der WT
      End_Ziel_QT_Pos : USInt;   // Position die ein verwendeter QT anfahren muß
      KorrPend : Real;   // Korrekturfaktor Pendelzeit
      KorrATZ : Real;   // Korrekturfaktor Abtropfzeit
      P_PNTER : Int;   // Parameter-Pointer
      B_PNTER : Int;   // Befehls-pointer
      SaveExpo : DInt;   // gerettete Expozeit bei Zwangsräumung
      Bereichstakte : USInt;   // Takt die der WT noch im aktuellen Behandlungsbereich verbringen muß
      Variante1 : Byte;
      Variante2 : Byte;
      Variante3 : Byte;
      Variante4 : Byte;
      Variante5 : Byte;
      akt_Ziel : Int;   // aktuelles Ziel aus FB9(FC120)
      akt_CMD : Byte;   // aktueller Befehl
      WT_Kennung : Byte;   // farbliche Markierung für PC
      Speed_Up : Int;
      Speed_Dn : Int;
      Speed_Fahrt : Int;
      resI : Int;
      Aufgabezeitpunkt : DInt;   // Systemzeit PC, wann WT aufgegeben wurde
      RestTakte : Int;   // Resttakte durch die Anlage
      "Name" : String[100];
      Befehl : Array[1..20] of Struct   // * Feldlänge anpassen DB45 beachten!!
         Kennung : Byte;   // Befehlskennung
         Startpos : Byte;   // Position
         Laenge : Byte;   // Länge
         Startpos2 : Byte;
         Laenge2 : Byte;
         Sonderparam : Byte;
         Param_Ptr : Int;   // Pointer für Parameter
      END_STRUCT;
      Param_Bereich : Array[1..100] of Byte;   // * Feldlänge anpassen DB45 beachten!!
   END_VAR
BEGIN
END_DATA_BLOCK

DATA_BLOCK "DB_WT11"   // DB111
{ S7_Optimized_Access := 'FALSE' }
AUTHOR : MS
// stored: AutoNumber false
   VAR RETAIN
      ANZAHL : Int := 10;   // * max. Anzahl der Befehle DB45 beachten!!
      OFFSET : Int := 180;   // * Beginn der Befehlskette
      LENG : Int := 8;   // * Befehlslänge in Byte
      WT_NR_lang : DInt;   // Warenträger-Nr. lang
      Oberflaeche : Real;   // Oberfläche in dm²
      Korb_Nr : USInt;   // Korbnummer (fest)
      POS : USInt;   // aktuelle Position
      Technologie : Int;   // Technologie Code
      priorisiert : Bool;   // WT ist proorisiert
      in_Anlage : Bool;   // will in die Anlage
      in_Entm : Bool;   // will in die Entmetallisierung
      aus_Anlage : Bool;   // kommt aus der Anlage
      aus_Entm : Bool;   // kommt aus der Entmetallisierung
      Speicher : Bool;   // Speicherprogramm
      FW_Pos : Bool;   // WT befindet sich am FW
      QT_Pos : Bool;   // WT befindet sich im QT
      Auto_Pos : USInt;   // Position für Automatikbetrieb
      Trommel : Bool;   // WT ist eine Trommel
      UT_Anforderung : Bool;   // Trockneranforderung erzeugt aus Befehl"FF"
      Stop : Bool;   // Stopbefehl aktiv
      Nassware : Bool;   // Nassware-Trichter am Entladestand anfordern
      TW_Pos : Bool;   // Warenträger ist noch in seiner Taktwechselposition
      noKorrBefx : Bool;   // Befehlsindex nicht korregieren
      noOPT_WT : Bool;   // kann nicht wie berechnet eingefahren werden
      last_Auto : Bool;   // letzter Umsetzvorgang erfolgte in Automatik
      Ziel_Pos_WT : USInt;   // Zielposition des WT für Korrektur beim Einsetzen
      lngsm_senken : Bool;   // langsam Senken
      lngsm_heben : Bool;   // langsam Heben
      lngsm_Fahrt : Bool;   // langsam Fahren
      WT_nok : Bool;   // Behandlungsfehler
      WT_151 : Bool;
      WT_161 : Bool;
      res226 : Bool;
      res227 : Bool;
      Alt_Befx : USInt;   // Befehlsindex in letzter Automatikposition
      Alt_Bereichstakte : USInt;   // Bereichstakte der letzten Automatikposition
      Alt_TW_Pos : USInt;
      Alt_Verweil : DInt;   // Verweilzeit der letzten Automatikposition
      Fertigzeitpunkt : DInt;   // Systemzeit PC, wann WT voraussichtlich fertig
      Meld_Pos : USInt;   // gemerkte Kollisionposition
      WT_Typ : Byte;   // Warenträgertyp (für die Zuordnung bestimmter Ware)
      End_Ziel_Pos : USInt;   // Zielposition an die der WT
      End_Ziel_QT_Pos : USInt;   // Position die ein verwendeter QT anfahren muß
      KorrPend : Real;   // Korrekturfaktor Pendelzeit
      KorrATZ : Real;   // Korrekturfaktor Abtropfzeit
      P_PNTER : Int;   // Parameter-Pointer
      B_PNTER : Int;   // Befehls-pointer
      SaveExpo : DInt;   // gerettete Expozeit bei Zwangsräumung
      Bereichstakte : USInt;   // Takt die der WT noch im aktuellen Behandlungsbereich verbringen muß
      Variante1 : Byte;
      Variante2 : Byte;
      Variante3 : Byte;
      Variante4 : Byte;
      Variante5 : Byte;
      akt_Ziel : Int;   // aktuelles Ziel aus FB9(FC120)
      akt_CMD : Byte;   // aktueller Befehl
      WT_Kennung : Byte;   // farbliche Markierung für PC
      Speed_Up : Int;
      Speed_Dn : Int;
      Speed_Fahrt : Int;
      resI : Int;
      Aufgabezeitpunkt : DInt;   // Systemzeit PC, wann WT aufgegeben wurde
      RestTakte : Int;   // Resttakte durch die Anlage
      "Name" : String[100];
      Befehl : Array[1..20] of Struct   // * Feldlänge anpassen DB45 beachten!!
         Kennung : Byte;   // Befehlskennung
         Startpos : Byte;   // Position
         Laenge : Byte;   // Länge
         Startpos2 : Byte;
         Laenge2 : Byte;
         Sonderparam : Byte;
         Param_Ptr : Int;   // Pointer für Parameter
      END_STRUCT;
      Param_Bereich : Array[1..100] of Byte;   // * Feldlänge anpassen DB45 beachten!!
   END_VAR
BEGIN
END_DATA_BLOCK

DATA_BLOCK "DB_WT12"   // DB112
{ S7_Optimized_Access := 'FALSE' }
AUTHOR : MS
// stored: AutoNumber false
   VAR RETAIN
      ANZAHL : Int := 10;   // * max. Anzahl der Befehle DB45 beachten!!
      OFFSET : Int := 180;   // * Beginn der Befehlskette
      LENG : Int := 8;   // * Befehlslänge in Byte
      WT_NR_lang : DInt;   // Warenträger-Nr. lang
      Oberflaeche : Real;   // Oberfläche in dm²
      Korb_Nr : USInt;   // Korbnummer (fest)
      POS : USInt;   // aktuelle Position
      Technologie : Int;   // Technologie Code
      priorisiert : Bool;   // WT ist proorisiert
      in_Anlage : Bool;   // will in die Anlage
      in_Entm : Bool;   // will in die Entmetallisierung
      aus_Anlage : Bool;   // kommt aus der Anlage
      aus_Entm : Bool;   // kommt aus der Entmetallisierung
      Speicher : Bool;   // Speicherprogramm
      FW_Pos : Bool;   // WT befindet sich am FW
      QT_Pos : Bool;   // WT befindet sich im QT
      Auto_Pos : USInt;   // Position für Automatikbetrieb
      Trommel : Bool;   // WT ist eine Trommel
      UT_Anforderung : Bool;   // Trockneranforderung erzeugt aus Befehl"FF"
      Stop : Bool;   // Stopbefehl aktiv
      Nassware : Bool;   // Nassware-Trichter am Entladestand anfordern
      TW_Pos : Bool;   // Warenträger ist noch in seiner Taktwechselposition
      noKorrBefx : Bool;   // Befehlsindex nicht korregieren
      noOPT_WT : Bool;   // kann nicht wie berechnet eingefahren werden
      last_Auto : Bool;   // letzter Umsetzvorgang erfolgte in Automatik
      Ziel_Pos_WT : USInt;   // Zielposition des WT für Korrektur beim Einsetzen
      lngsm_senken : Bool;   // langsam Senken
      lngsm_heben : Bool;   // langsam Heben
      lngsm_Fahrt : Bool;   // langsam Fahren
      WT_nok : Bool;   // Behandlungsfehler
      WT_151 : Bool;
      WT_161 : Bool;
      res226 : Bool;
      res227 : Bool;
      Alt_Befx : USInt;   // Befehlsindex in letzter Automatikposition
      Alt_Bereichstakte : USInt;   // Bereichstakte der letzten Automatikposition
      Alt_TW_Pos : USInt;
      Alt_Verweil : DInt;   // Verweilzeit der letzten Automatikposition
      Fertigzeitpunkt : DInt;   // Systemzeit PC, wann WT voraussichtlich fertig
      Meld_Pos : USInt;   // gemerkte Kollisionposition
      WT_Typ : Byte;   // Warenträgertyp (für die Zuordnung bestimmter Ware)
      End_Ziel_Pos : USInt;   // Zielposition an die der WT
      End_Ziel_QT_Pos : USInt;   // Position die ein verwendeter QT anfahren muß
      KorrPend : Real;   // Korrekturfaktor Pendelzeit
      KorrATZ : Real;   // Korrekturfaktor Abtropfzeit
      P_PNTER : Int;   // Parameter-Pointer
      B_PNTER : Int;   // Befehls-pointer
      SaveExpo : DInt;   // gerettete Expozeit bei Zwangsräumung
      Bereichstakte : USInt;   // Takt die der WT noch im aktuellen Behandlungsbereich verbringen muß
      Variante1 : Byte;
      Variante2 : Byte;
      Variante3 : Byte;
      Variante4 : Byte;
      Variante5 : Byte;
      akt_Ziel : Int;   // aktuelles Ziel aus FB9(FC120)
      akt_CMD : Byte;   // aktueller Befehl
      WT_Kennung : Byte;   // farbliche Markierung für PC
      Speed_Up : Int;
      Speed_Dn : Int;
      Speed_Fahrt : Int;
      resI : Int;
      Aufgabezeitpunkt : DInt;   // Systemzeit PC, wann WT aufgegeben wurde
      RestTakte : Int;   // Resttakte durch die Anlage
      "Name" : String[100];
      Befehl : Array[1..20] of Struct   // * Feldlänge anpassen DB45 beachten!!
         Kennung : Byte;   // Befehlskennung
         Startpos : Byte;   // Position
         Laenge : Byte;   // Länge
         Startpos2 : Byte;
         Laenge2 : Byte;
         Sonderparam : Byte;
         Param_Ptr : Int;   // Pointer für Parameter
      END_STRUCT;
      Param_Bereich : Array[1..100] of Byte;   // * Feldlänge anpassen DB45 beachten!!
   END_VAR
BEGIN
END_DATA_BLOCK

DATA_BLOCK "DB_WT2"   // DB102
{ S7_Optimized_Access := 'FALSE' }
AUTHOR : MS
// stored: AutoNumber false
   VAR RETAIN
      ANZAHL : Int := 10;   // * max. Anzahl der Befehle DB45 beachten!!
      OFFSET : Int := 180;   // * Beginn der Befehlskette
      LENG : Int := 8;   // * Befehlslänge in Byte
      WT_NR_lang : DInt;   // Warenträger-Nr. lang
      Oberflaeche : Real;   // Oberfläche in dm²
      Korb_Nr : USInt;   // Korbnummer (fest)
      POS : USInt;   // aktuelle Position
      Technologie : Int;   // Technologie Code
      priorisiert : Bool;   // WT ist proorisiert
      in_Anlage : Bool;   // will in die Anlage
      in_Entm : Bool;   // will in die Entmetallisierung
      aus_Anlage : Bool;   // kommt aus der Anlage
      aus_Entm : Bool;   // kommt aus der Entmetallisierung
      Speicher : Bool;   // Speicherprogramm
      FW_Pos : Bool;   // WT befindet sich am FW
      QT_Pos : Bool;   // WT befindet sich im QT
      Auto_Pos : USInt;   // Position für Automatikbetrieb
      Trommel : Bool;   // WT ist eine Trommel
      UT_Anforderung : Bool;   // Trockneranforderung erzeugt aus Befehl"FF"
      Stop : Bool;   // Stopbefehl aktiv
      Nassware : Bool;   // Nassware-Trichter am Entladestand anfordern
      TW_Pos : Bool;   // Warenträger ist noch in seiner Taktwechselposition
      noKorrBefx : Bool;   // Befehlsindex nicht korregieren
      noOPT_WT : Bool;   // kann nicht wie berechnet eingefahren werden
      last_Auto : Bool;   // letzter Umsetzvorgang erfolgte in Automatik
      Ziel_Pos_WT : USInt;   // Zielposition des WT für Korrektur beim Einsetzen
      lngsm_senken : Bool;   // langsam Senken
      lngsm_heben : Bool;   // langsam Heben
      lngsm_Fahrt : Bool;   // langsam Fahren
      WT_nok : Bool;   // Behandlungsfehler
      WT_151 : Bool;
      WT_161 : Bool;
      res226 : Bool;
      res227 : Bool;
      Alt_Befx : USInt;   // Befehlsindex in letzter Automatikposition
      Alt_Bereichstakte : USInt;   // Bereichstakte der letzten Automatikposition
      Alt_TW_Pos : USInt;
      Alt_Verweil : DInt;   // Verweilzeit der letzten Automatikposition
      Fertigzeitpunkt : DInt;   // Systemzeit PC, wann WT voraussichtlich fertig
      Meld_Pos : USInt;   // gemerkte Kollisionposition
      WT_Typ : Byte;   // Warenträgertyp (für die Zuordnung bestimmter Ware)
      End_Ziel_Pos : USInt;   // Zielposition an die der WT
      End_Ziel_QT_Pos : USInt;   // Position die ein verwendeter QT anfahren muß
      KorrPend : Real;   // Korrekturfaktor Pendelzeit
      KorrATZ : Real;   // Korrekturfaktor Abtropfzeit
      P_PNTER : Int;   // Parameter-Pointer
      B_PNTER : Int;   // Befehls-pointer
      SaveExpo : DInt;   // gerettete Expozeit bei Zwangsräumung
      Bereichstakte : USInt;   // Takt die der WT noch im aktuellen Behandlungsbereich verbringen muß
      Variante1 : Byte;
      Variante2 : Byte;
      Variante3 : Byte;
      Variante4 : Byte;
      Variante5 : Byte;
      akt_Ziel : Int;   // aktuelles Ziel aus FB9(FC120)
      akt_CMD : Byte;   // aktueller Befehl
      WT_Kennung : Byte;   // farbliche Markierung für PC
      Speed_Up : Int;
      Speed_Dn : Int;
      Speed_Fahrt : Int;
      resI : Int;
      Aufgabezeitpunkt : DInt;   // Systemzeit PC, wann WT aufgegeben wurde
      RestTakte : Int;   // Resttakte durch die Anlage
      "Name" : String[100];
      Befehl : Array[1..20] of Struct   // * Feldlänge anpassen DB45 beachten!!
         Kennung : Byte;   // Befehlskennung
         Startpos : Byte;   // Position
         Laenge : Byte;   // Länge
         Startpos2 : Byte;
         Laenge2 : Byte;
         Sonderparam : Byte;
         Param_Ptr : Int;   // Pointer für Parameter
      END_STRUCT;
      Param_Bereich : Array[1..100] of Byte;   // * Feldlänge anpassen DB45 beachten!!
   END_VAR
BEGIN
END_DATA_BLOCK

DATA_BLOCK "DB_WT3"   // DB103
{ S7_Optimized_Access := 'FALSE' }
AUTHOR : MS
// stored: AutoNumber false
   VAR RETAIN
      ANZAHL : Int := 10;   // * max. Anzahl der Befehle DB45 beachten!!
      OFFSET : Int := 180;   // * Beginn der Befehlskette
      LENG : Int := 8;   // * Befehlslänge in Byte
      WT_NR_lang : DInt;   // Warenträger-Nr. lang
      Oberflaeche : Real;   // Oberfläche in dm²
      Korb_Nr : USInt;   // Korbnummer (fest)
      POS : USInt;   // aktuelle Position
      Technologie : Int;   // Technologie Code
      priorisiert : Bool;   // WT ist proorisiert
      in_Anlage : Bool;   // will in die Anlage
      in_Entm : Bool;   // will in die Entmetallisierung
      aus_Anlage : Bool;   // kommt aus der Anlage
      aus_Entm : Bool;   // kommt aus der Entmetallisierung
      Speicher : Bool;   // Speicherprogramm
      FW_Pos : Bool;   // WT befindet sich am FW
      QT_Pos : Bool;   // WT befindet sich im QT
      Auto_Pos : USInt;   // Position für Automatikbetrieb
      Trommel : Bool;   // WT ist eine Trommel
      UT_Anforderung : Bool;   // Trockneranforderung erzeugt aus Befehl"FF"
      Stop : Bool;   // Stopbefehl aktiv
      Nassware : Bool;   // Nassware-Trichter am Entladestand anfordern
      TW_Pos : Bool;   // Warenträger ist noch in seiner Taktwechselposition
      noKorrBefx : Bool;   // Befehlsindex nicht korregieren
      noOPT_WT : Bool;   // kann nicht wie berechnet eingefahren werden
      last_Auto : Bool;   // letzter Umsetzvorgang erfolgte in Automatik
      Ziel_Pos_WT : USInt;   // Zielposition des WT für Korrektur beim Einsetzen
      lngsm_senken : Bool;   // langsam Senken
      lngsm_heben : Bool;   // langsam Heben
      lngsm_Fahrt : Bool;   // langsam Fahren
      WT_nok : Bool;   // Behandlungsfehler
      WT_151 : Bool;
      WT_161 : Bool;
      res226 : Bool;
      res227 : Bool;
      Alt_Befx : USInt;   // Befehlsindex in letzter Automatikposition
      Alt_Bereichstakte : USInt;   // Bereichstakte der letzten Automatikposition
      Alt_TW_Pos : USInt;
      Alt_Verweil : DInt;   // Verweilzeit der letzten Automatikposition
      Fertigzeitpunkt : DInt;   // Systemzeit PC, wann WT voraussichtlich fertig
      Meld_Pos : USInt;   // gemerkte Kollisionposition
      WT_Typ : Byte;   // Warenträgertyp (für die Zuordnung bestimmter Ware)
      End_Ziel_Pos : USInt;   // Zielposition an die der WT
      End_Ziel_QT_Pos : USInt;   // Position die ein verwendeter QT anfahren muß
      KorrPend : Real;   // Korrekturfaktor Pendelzeit
      KorrATZ : Real;   // Korrekturfaktor Abtropfzeit
      P_PNTER : Int;   // Parameter-Pointer
      B_PNTER : Int;   // Befehls-pointer
      SaveExpo : DInt;   // gerettete Expozeit bei Zwangsräumung
      Bereichstakte : USInt;   // Takt die der WT noch im aktuellen Behandlungsbereich verbringen muß
      Variante1 : Byte;
      Variante2 : Byte;
      Variante3 : Byte;
      Variante4 : Byte;
      Variante5 : Byte;
      akt_Ziel : Int;   // aktuelles Ziel aus FB9(FC120)
      akt_CMD : Byte;   // aktueller Befehl
      WT_Kennung : Byte;   // farbliche Markierung für PC
      Speed_Up : Int;
      Speed_Dn : Int;
      Speed_Fahrt : Int;
      resI : Int;
      Aufgabezeitpunkt : DInt;   // Systemzeit PC, wann WT aufgegeben wurde
      RestTakte : Int;   // Resttakte durch die Anlage
      "Name" : String[100];
      Befehl : Array[1..20] of Struct   // * Feldlänge anpassen DB45 beachten!!
         Kennung : Byte;   // Befehlskennung
         Startpos : Byte;   // Position
         Laenge : Byte;   // Länge
         Startpos2 : Byte;
         Laenge2 : Byte;
         Sonderparam : Byte;
         Param_Ptr : Int;   // Pointer für Parameter
      END_STRUCT;
      Param_Bereich : Array[1..100] of Byte;   // * Feldlänge anpassen DB45 beachten!!
   END_VAR
BEGIN
END_DATA_BLOCK

DATA_BLOCK "DB_WT4"   // DB104
{ S7_Optimized_Access := 'FALSE' }
AUTHOR : MS
// stored: AutoNumber false
   VAR RETAIN
      ANZAHL : Int := 10;   // * max. Anzahl der Befehle DB45 beachten!!
      OFFSET : Int := 180;   // * Beginn der Befehlskette
      LENG : Int := 8;   // * Befehlslänge in Byte
      WT_NR_lang : DInt;   // Warenträger-Nr. lang
      Oberflaeche : Real;   // Oberfläche in dm²
      Korb_Nr : USInt;   // Korbnummer (fest)
      POS : USInt;   // aktuelle Position
      Technologie : Int;   // Technologie Code
      priorisiert : Bool;   // WT ist proorisiert
      in_Anlage : Bool;   // will in die Anlage
      in_Entm : Bool;   // will in die Entmetallisierung
      aus_Anlage : Bool;   // kommt aus der Anlage
      aus_Entm : Bool;   // kommt aus der Entmetallisierung
      Speicher : Bool;   // Speicherprogramm
      FW_Pos : Bool;   // WT befindet sich am FW
      QT_Pos : Bool;   // WT befindet sich im QT
      Auto_Pos : USInt;   // Position für Automatikbetrieb
      Trommel : Bool;   // WT ist eine Trommel
      UT_Anforderung : Bool;   // Trockneranforderung erzeugt aus Befehl"FF"
      Stop : Bool;   // Stopbefehl aktiv
      Nassware : Bool;   // Nassware-Trichter am Entladestand anfordern
      TW_Pos : Bool;   // Warenträger ist noch in seiner Taktwechselposition
      noKorrBefx : Bool;   // Befehlsindex nicht korregieren
      noOPT_WT : Bool;   // kann nicht wie berechnet eingefahren werden
      last_Auto : Bool;   // letzter Umsetzvorgang erfolgte in Automatik
      Ziel_Pos_WT : USInt;   // Zielposition des WT für Korrektur beim Einsetzen
      lngsm_senken : Bool;   // langsam Senken
      lngsm_heben : Bool;   // langsam Heben
      lngsm_Fahrt : Bool;   // langsam Fahren
      WT_nok : Bool;   // Behandlungsfehler
      WT_151 : Bool;
      WT_161 : Bool;
      res226 : Bool;
      res227 : Bool;
      Alt_Befx : USInt;   // Befehlsindex in letzter Automatikposition
      Alt_Bereichstakte : USInt;   // Bereichstakte der letzten Automatikposition
      Alt_TW_Pos : USInt;
      Alt_Verweil : DInt;   // Verweilzeit der letzten Automatikposition
      Fertigzeitpunkt : DInt;   // Systemzeit PC, wann WT voraussichtlich fertig
      Meld_Pos : USInt;   // gemerkte Kollisionposition
      WT_Typ : Byte;   // Warenträgertyp (für die Zuordnung bestimmter Ware)
      End_Ziel_Pos : USInt;   // Zielposition an die der WT
      End_Ziel_QT_Pos : USInt;   // Position die ein verwendeter QT anfahren muß
      KorrPend : Real;   // Korrekturfaktor Pendelzeit
      KorrATZ : Real;   // Korrekturfaktor Abtropfzeit
      P_PNTER : Int;   // Parameter-Pointer
      B_PNTER : Int;   // Befehls-pointer
      SaveExpo : DInt;   // gerettete Expozeit bei Zwangsräumung
      Bereichstakte : USInt;   // Takt die der WT noch im aktuellen Behandlungsbereich verbringen muß
      Variante1 : Byte;
      Variante2 : Byte;
      Variante3 : Byte;
      Variante4 : Byte;
      Variante5 : Byte;
      akt_Ziel : Int;   // aktuelles Ziel aus FB9(FC120)
      akt_CMD : Byte;   // aktueller Befehl
      WT_Kennung : Byte;   // farbliche Markierung für PC
      Speed_Up : Int;
      Speed_Dn : Int;
      Speed_Fahrt : Int;
      resI : Int;
      Aufgabezeitpunkt : DInt;   // Systemzeit PC, wann WT aufgegeben wurde
      RestTakte : Int;   // Resttakte durch die Anlage
      "Name" : String[100];
      Befehl : Array[1..20] of Struct   // * Feldlänge anpassen DB45 beachten!!
         Kennung : Byte;   // Befehlskennung
         Startpos : Byte;   // Position
         Laenge : Byte;   // Länge
         Startpos2 : Byte;
         Laenge2 : Byte;
         Sonderparam : Byte;
         Param_Ptr : Int;   // Pointer für Parameter
      END_STRUCT;
      Param_Bereich : Array[1..100] of Byte;   // * Feldlänge anpassen DB45 beachten!!
   END_VAR
BEGIN
END_DATA_BLOCK

DATA_BLOCK "DB_WT5"   // DB105
{ S7_Optimized_Access := 'FALSE' }
AUTHOR : MS
// stored: AutoNumber false
   VAR RETAIN
      ANZAHL : Int := 10;   // * max. Anzahl der Befehle DB45 beachten!!
      OFFSET : Int := 180;   // * Beginn der Befehlskette
      LENG : Int := 8;   // * Befehlslänge in Byte
      WT_NR_lang : DInt;   // Warenträger-Nr. lang
      Oberflaeche : Real;   // Oberfläche in dm²
      Korb_Nr : USInt;   // Korbnummer (fest)
      POS : USInt;   // aktuelle Position
      Technologie : Int;   // Technologie Code
      priorisiert : Bool;   // WT ist proorisiert
      in_Anlage : Bool;   // will in die Anlage
      in_Entm : Bool;   // will in die Entmetallisierung
      aus_Anlage : Bool;   // kommt aus der Anlage
      aus_Entm : Bool;   // kommt aus der Entmetallisierung
      Speicher : Bool;   // Speicherprogramm
      FW_Pos : Bool;   // WT befindet sich am FW
      QT_Pos : Bool;   // WT befindet sich im QT
      Auto_Pos : USInt;   // Position für Automatikbetrieb
      Trommel : Bool;   // WT ist eine Trommel
      UT_Anforderung : Bool;   // Trockneranforderung erzeugt aus Befehl"FF"
      Stop : Bool;   // Stopbefehl aktiv
      Nassware : Bool;   // Nassware-Trichter am Entladestand anfordern
      TW_Pos : Bool;   // Warenträger ist noch in seiner Taktwechselposition
      noKorrBefx : Bool;   // Befehlsindex nicht korregieren
      noOPT_WT : Bool;   // kann nicht wie berechnet eingefahren werden
      last_Auto : Bool;   // letzter Umsetzvorgang erfolgte in Automatik
      Ziel_Pos_WT : USInt;   // Zielposition des WT für Korrektur beim Einsetzen
      lngsm_senken : Bool;   // langsam Senken
      lngsm_heben : Bool;   // langsam Heben
      lngsm_Fahrt : Bool;   // langsam Fahren
      WT_nok : Bool;   // Behandlungsfehler
      WT_151 : Bool;
      WT_161 : Bool;
      res226 : Bool;
      res227 : Bool;
      Alt_Befx : USInt;   // Befehlsindex in letzter Automatikposition
      Alt_Bereichstakte : USInt;   // Bereichstakte der letzten Automatikposition
      Alt_TW_Pos : USInt;
      Alt_Verweil : DInt;   // Verweilzeit der letzten Automatikposition
      Fertigzeitpunkt : DInt;   // Systemzeit PC, wann WT voraussichtlich fertig
      Meld_Pos : USInt;   // gemerkte Kollisionposition
      WT_Typ : Byte;   // Warenträgertyp (für die Zuordnung bestimmter Ware)
      End_Ziel_Pos : USInt;   // Zielposition an die der WT
      End_Ziel_QT_Pos : USInt;   // Position die ein verwendeter QT anfahren muß
      KorrPend : Real;   // Korrekturfaktor Pendelzeit
      KorrATZ : Real;   // Korrekturfaktor Abtropfzeit
      P_PNTER : Int;   // Parameter-Pointer
      B_PNTER : Int;   // Befehls-pointer
      SaveExpo : DInt;   // gerettete Expozeit bei Zwangsräumung
      Bereichstakte : USInt;   // Takt die der WT noch im aktuellen Behandlungsbereich verbringen muß
      Variante1 : Byte;
      Variante2 : Byte;
      Variante3 : Byte;
      Variante4 : Byte;
      Variante5 : Byte;
      akt_Ziel : Int;   // aktuelles Ziel aus FB9(FC120)
      akt_CMD : Byte;   // aktueller Befehl
      WT_Kennung : Byte;   // farbliche Markierung für PC
      Speed_Up : Int;
      Speed_Dn : Int;
      Speed_Fahrt : Int;
      resI : Int;
      Aufgabezeitpunkt : DInt;   // Systemzeit PC, wann WT aufgegeben wurde
      RestTakte : Int;   // Resttakte durch die Anlage
      "Name" : String[100];
      Befehl : Array[1..20] of Struct   // * Feldlänge anpassen DB45 beachten!!
         Kennung : Byte;   // Befehlskennung
         Startpos : Byte;   // Position
         Laenge : Byte;   // Länge
         Startpos2 : Byte;
         Laenge2 : Byte;
         Sonderparam : Byte;
         Param_Ptr : Int;   // Pointer für Parameter
      END_STRUCT;
      Param_Bereich : Array[1..100] of Byte;   // * Feldlänge anpassen DB45 beachten!!
   END_VAR
BEGIN
END_DATA_BLOCK

DATA_BLOCK "DB_WT6"   // DB106
{ S7_Optimized_Access := 'FALSE' }
AUTHOR : MS
// stored: AutoNumber false
   VAR RETAIN
      ANZAHL : Int := 10;   // * max. Anzahl der Befehle DB45 beachten!!
      OFFSET : Int := 180;   // * Beginn der Befehlskette
      LENG : Int := 8;   // * Befehlslänge in Byte
      WT_NR_lang : DInt;   // Warenträger-Nr. lang
      Oberflaeche : Real;   // Oberfläche in dm²
      Korb_Nr : USInt;   // Korbnummer (fest)
      POS : USInt;   // aktuelle Position
      Technologie : Int;   // Technologie Code
      priorisiert : Bool;   // WT ist proorisiert
      in_Anlage : Bool;   // will in die Anlage
      in_Entm : Bool;   // will in die Entmetallisierung
      aus_Anlage : Bool;   // kommt aus der Anlage
      aus_Entm : Bool;   // kommt aus der Entmetallisierung
      Speicher : Bool;   // Speicherprogramm
      FW_Pos : Bool;   // WT befindet sich am FW
      QT_Pos : Bool;   // WT befindet sich im QT
      Auto_Pos : USInt;   // Position für Automatikbetrieb
      Trommel : Bool;   // WT ist eine Trommel
      UT_Anforderung : Bool;   // Trockneranforderung erzeugt aus Befehl"FF"
      Stop : Bool;   // Stopbefehl aktiv
      Nassware : Bool;   // Nassware-Trichter am Entladestand anfordern
      TW_Pos : Bool;   // Warenträger ist noch in seiner Taktwechselposition
      noKorrBefx : Bool;   // Befehlsindex nicht korregieren
      noOPT_WT : Bool;   // kann nicht wie berechnet eingefahren werden
      last_Auto : Bool;   // letzter Umsetzvorgang erfolgte in Automatik
      Ziel_Pos_WT : USInt;   // Zielposition des WT für Korrektur beim Einsetzen
      lngsm_senken : Bool;   // langsam Senken
      lngsm_heben : Bool;   // langsam Heben
      lngsm_Fahrt : Bool;   // langsam Fahren
      WT_nok : Bool;   // Behandlungsfehler
      WT_151 : Bool;
      WT_161 : Bool;
      res226 : Bool;
      res227 : Bool;
      Alt_Befx : USInt;   // Befehlsindex in letzter Automatikposition
      Alt_Bereichstakte : USInt;   // Bereichstakte der letzten Automatikposition
      Alt_TW_Pos : USInt;
      Alt_Verweil : DInt;   // Verweilzeit der letzten Automatikposition
      Fertigzeitpunkt : DInt;   // Systemzeit PC, wann WT voraussichtlich fertig
      Meld_Pos : USInt;   // gemerkte Kollisionposition
      WT_Typ : Byte;   // Warenträgertyp (für die Zuordnung bestimmter Ware)
      End_Ziel_Pos : USInt;   // Zielposition an die der WT
      End_Ziel_QT_Pos : USInt;   // Position die ein verwendeter QT anfahren muß
      KorrPend : Real;   // Korrekturfaktor Pendelzeit
      KorrATZ : Real;   // Korrekturfaktor Abtropfzeit
      P_PNTER : Int;   // Parameter-Pointer
      B_PNTER : Int;   // Befehls-pointer
      SaveExpo : DInt;   // gerettete Expozeit bei Zwangsräumung
      Bereichstakte : USInt;   // Takt die der WT noch im aktuellen Behandlungsbereich verbringen muß
      Variante1 : Byte;
      Variante2 : Byte;
      Variante3 : Byte;
      Variante4 : Byte;
      Variante5 : Byte;
      akt_Ziel : Int;   // aktuelles Ziel aus FB9(FC120)
      akt_CMD : Byte;   // aktueller Befehl
      WT_Kennung : Byte;   // farbliche Markierung für PC
      Speed_Up : Int;
      Speed_Dn : Int;
      Speed_Fahrt : Int;
      resI : Int;
      Aufgabezeitpunkt : DInt;   // Systemzeit PC, wann WT aufgegeben wurde
      RestTakte : Int;   // Resttakte durch die Anlage
      "Name" : String[100];
      Befehl : Array[1..20] of Struct   // * Feldlänge anpassen DB45 beachten!!
         Kennung : Byte;   // Befehlskennung
         Startpos : Byte;   // Position
         Laenge : Byte;   // Länge
         Startpos2 : Byte;
         Laenge2 : Byte;
         Sonderparam : Byte;
         Param_Ptr : Int;   // Pointer für Parameter
      END_STRUCT;
      Param_Bereich : Array[1..100] of Byte;   // * Feldlänge anpassen DB45 beachten!!
   END_VAR
BEGIN
END_DATA_BLOCK

DATA_BLOCK "DB_WT7"   // DB107
{ S7_Optimized_Access := 'FALSE' }
AUTHOR : MS
// stored: AutoNumber false
   VAR RETAIN
      ANZAHL : Int := 10;   // * max. Anzahl der Befehle DB45 beachten!!
      OFFSET : Int := 180;   // * Beginn der Befehlskette
      LENG : Int := 8;   // * Befehlslänge in Byte
      WT_NR_lang : DInt;   // Warenträger-Nr. lang
      Oberflaeche : Real;   // Oberfläche in dm²
      Korb_Nr : USInt;   // Korbnummer (fest)
      POS : USInt;   // aktuelle Position
      Technologie : Int;   // Technologie Code
      priorisiert : Bool;   // WT ist proorisiert
      in_Anlage : Bool;   // will in die Anlage
      in_Entm : Bool;   // will in die Entmetallisierung
      aus_Anlage : Bool;   // kommt aus der Anlage
      aus_Entm : Bool;   // kommt aus der Entmetallisierung
      Speicher : Bool;   // Speicherprogramm
      FW_Pos : Bool;   // WT befindet sich am FW
      QT_Pos : Bool;   // WT befindet sich im QT
      Auto_Pos : USInt;   // Position für Automatikbetrieb
      Trommel : Bool;   // WT ist eine Trommel
      UT_Anforderung : Bool;   // Trockneranforderung erzeugt aus Befehl"FF"
      Stop : Bool;   // Stopbefehl aktiv
      Nassware : Bool;   // Nassware-Trichter am Entladestand anfordern
      TW_Pos : Bool;   // Warenträger ist noch in seiner Taktwechselposition
      noKorrBefx : Bool;   // Befehlsindex nicht korregieren
      noOPT_WT : Bool;   // kann nicht wie berechnet eingefahren werden
      last_Auto : Bool;   // letzter Umsetzvorgang erfolgte in Automatik
      Ziel_Pos_WT : USInt;   // Zielposition des WT für Korrektur beim Einsetzen
      lngsm_senken : Bool;   // langsam Senken
      lngsm_heben : Bool;   // langsam Heben
      lngsm_Fahrt : Bool;   // langsam Fahren
      WT_nok : Bool;   // Behandlungsfehler
      WT_151 : Bool;
      WT_161 : Bool;
      res226 : Bool;
      res227 : Bool;
      Alt_Befx : USInt;   // Befehlsindex in letzter Automatikposition
      Alt_Bereichstakte : USInt;   // Bereichstakte der letzten Automatikposition
      Alt_TW_Pos : USInt;
      Alt_Verweil : DInt;   // Verweilzeit der letzten Automatikposition
      Fertigzeitpunkt : DInt;   // Systemzeit PC, wann WT voraussichtlich fertig
      Meld_Pos : USInt;   // gemerkte Kollisionposition
      WT_Typ : Byte;   // Warenträgertyp (für die Zuordnung bestimmter Ware)
      End_Ziel_Pos : USInt;   // Zielposition an die der WT
      End_Ziel_QT_Pos : USInt;   // Position die ein verwendeter QT anfahren muß
      KorrPend : Real;   // Korrekturfaktor Pendelzeit
      KorrATZ : Real;   // Korrekturfaktor Abtropfzeit
      P_PNTER : Int;   // Parameter-Pointer
      B_PNTER : Int;   // Befehls-pointer
      SaveExpo : DInt;   // gerettete Expozeit bei Zwangsräumung
      Bereichstakte : USInt;   // Takt die der WT noch im aktuellen Behandlungsbereich verbringen muß
      Variante1 : Byte;
      Variante2 : Byte;
      Variante3 : Byte;
      Variante4 : Byte;
      Variante5 : Byte;
      akt_Ziel : Int;   // aktuelles Ziel aus FB9(FC120)
      akt_CMD : Byte;   // aktueller Befehl
      WT_Kennung : Byte;   // farbliche Markierung für PC
      Speed_Up : Int;
      Speed_Dn : Int;
      Speed_Fahrt : Int;
      resI : Int;
      Aufgabezeitpunkt : DInt;   // Systemzeit PC, wann WT aufgegeben wurde
      RestTakte : Int;   // Resttakte durch die Anlage
      "Name" : String[100];
      Befehl : Array[1..20] of Struct   // * Feldlänge anpassen DB45 beachten!!
         Kennung : Byte;   // Befehlskennung
         Startpos : Byte;   // Position
         Laenge : Byte;   // Länge
         Startpos2 : Byte;
         Laenge2 : Byte;
         Sonderparam : Byte;
         Param_Ptr : Int;   // Pointer für Parameter
      END_STRUCT;
      Param_Bereich : Array[1..100] of Byte;   // * Feldlänge anpassen DB45 beachten!!
   END_VAR
BEGIN
END_DATA_BLOCK

DATA_BLOCK "DB_WT8"   // DB108
{ S7_Optimized_Access := 'FALSE' }
AUTHOR : MS
// stored: AutoNumber false
   VAR RETAIN
      ANZAHL : Int := 10;   // * max. Anzahl der Befehle DB45 beachten!!
      OFFSET : Int := 180;   // * Beginn der Befehlskette
      LENG : Int := 8;   // * Befehlslänge in Byte
      WT_NR_lang : DInt;   // Warenträger-Nr. lang
      Oberflaeche : Real;   // Oberfläche in dm²
      Korb_Nr : USInt;   // Korbnummer (fest)
      POS : USInt;   // aktuelle Position
      Technologie : Int;   // Technologie Code
      priorisiert : Bool;   // WT ist proorisiert
      in_Anlage : Bool;   // will in die Anlage
      in_Entm : Bool;   // will in die Entmetallisierung
      aus_Anlage : Bool;   // kommt aus der Anlage
      aus_Entm : Bool;   // kommt aus der Entmetallisierung
      Speicher : Bool;   // Speicherprogramm
      FW_Pos : Bool;   // WT befindet sich am FW
      QT_Pos : Bool;   // WT befindet sich im QT
      Auto_Pos : USInt;   // Position für Automatikbetrieb
      Trommel : Bool;   // WT ist eine Trommel
      UT_Anforderung : Bool;   // Trockneranforderung erzeugt aus Befehl"FF"
      Stop : Bool;   // Stopbefehl aktiv
      Nassware : Bool;   // Nassware-Trichter am Entladestand anfordern
      TW_Pos : Bool;   // Warenträger ist noch in seiner Taktwechselposition
      noKorrBefx : Bool;   // Befehlsindex nicht korregieren
      noOPT_WT : Bool;   // kann nicht wie berechnet eingefahren werden
      last_Auto : Bool;   // letzter Umsetzvorgang erfolgte in Automatik
      Ziel_Pos_WT : USInt;   // Zielposition des WT für Korrektur beim Einsetzen
      lngsm_senken : Bool;   // langsam Senken
      lngsm_heben : Bool;   // langsam Heben
      lngsm_Fahrt : Bool;   // langsam Fahren
      WT_nok : Bool;   // Behandlungsfehler
      WT_151 : Bool;
      WT_161 : Bool;
      res226 : Bool;
      res227 : Bool;
      Alt_Befx : USInt;   // Befehlsindex in letzter Automatikposition
      Alt_Bereichstakte : USInt;   // Bereichstakte der letzten Automatikposition
      Alt_TW_Pos : USInt;
      Alt_Verweil : DInt;   // Verweilzeit der letzten Automatikposition
      Fertigzeitpunkt : DInt;   // Systemzeit PC, wann WT voraussichtlich fertig
      Meld_Pos : USInt;   // gemerkte Kollisionposition
      WT_Typ : Byte;   // Warenträgertyp (für die Zuordnung bestimmter Ware)
      End_Ziel_Pos : USInt;   // Zielposition an die der WT
      End_Ziel_QT_Pos : USInt;   // Position die ein verwendeter QT anfahren muß
      KorrPend : Real;   // Korrekturfaktor Pendelzeit
      KorrATZ : Real;   // Korrekturfaktor Abtropfzeit
      P_PNTER : Int;   // Parameter-Pointer
      B_PNTER : Int;   // Befehls-pointer
      SaveExpo : DInt;   // gerettete Expozeit bei Zwangsräumung
      Bereichstakte : USInt;   // Takt die der WT noch im aktuellen Behandlungsbereich verbringen muß
      Variante1 : Byte;
      Variante2 : Byte;
      Variante3 : Byte;
      Variante4 : Byte;
      Variante5 : Byte;
      akt_Ziel : Int;   // aktuelles Ziel aus FB9(FC120)
      akt_CMD : Byte;   // aktueller Befehl
      WT_Kennung : Byte;   // farbliche Markierung für PC
      Speed_Up : Int;
      Speed_Dn : Int;
      Speed_Fahrt : Int;
      resI : Int;
      Aufgabezeitpunkt : DInt;   // Systemzeit PC, wann WT aufgegeben wurde
      RestTakte : Int;   // Resttakte durch die Anlage
      "Name" : String[100];
      Befehl : Array[1..20] of Struct   // * Feldlänge anpassen DB45 beachten!!
         Kennung : Byte;   // Befehlskennung
         Startpos : Byte;   // Position
         Laenge : Byte;   // Länge
         Startpos2 : Byte;
         Laenge2 : Byte;
         Sonderparam : Byte;
         Param_Ptr : Int;   // Pointer für Parameter
      END_STRUCT;
      Param_Bereich : Array[1..100] of Byte;   // * Feldlänge anpassen DB45 beachten!!
   END_VAR
BEGIN
END_DATA_BLOCK

DATA_BLOCK "DB_WT9"   // DB109
{ S7_Optimized_Access := 'FALSE' }
AUTHOR : MS
// stored: AutoNumber false
   VAR RETAIN
      ANZAHL : Int := 10;   // * max. Anzahl der Befehle DB45 beachten!!
      OFFSET : Int := 180;   // * Beginn der Befehlskette
      LENG : Int := 8;   // * Befehlslänge in Byte
      WT_NR_lang : DInt;   // Warenträger-Nr. lang
      Oberflaeche : Real;   // Oberfläche in dm²
      Korb_Nr : USInt;   // Korbnummer (fest)
      POS : USInt;   // aktuelle Position
      Technologie : Int;   // Technologie Code
      priorisiert : Bool;   // WT ist proorisiert
      in_Anlage : Bool;   // will in die Anlage
      in_Entm : Bool;   // will in die Entmetallisierung
      aus_Anlage : Bool;   // kommt aus der Anlage
      aus_Entm : Bool;   // kommt aus der Entmetallisierung
      Speicher : Bool;   // Speicherprogramm
      FW_Pos : Bool;   // WT befindet sich am FW
      QT_Pos : Bool;   // WT befindet sich im QT
      Auto_Pos : USInt;   // Position für Automatikbetrieb
      Trommel : Bool;   // WT ist eine Trommel
      UT_Anforderung : Bool;   // Trockneranforderung erzeugt aus Befehl"FF"
      Stop : Bool;   // Stopbefehl aktiv
      Nassware : Bool;   // Nassware-Trichter am Entladestand anfordern
      TW_Pos : Bool;   // Warenträger ist noch in seiner Taktwechselposition
      noKorrBefx : Bool;   // Befehlsindex nicht korregieren
      noOPT_WT : Bool;   // kann nicht wie berechnet eingefahren werden
      last_Auto : Bool;   // letzter Umsetzvorgang erfolgte in Automatik
      Ziel_Pos_WT : USInt;   // Zielposition des WT für Korrektur beim Einsetzen
      lngsm_senken : Bool;   // langsam Senken
      lngsm_heben : Bool;   // langsam Heben
      lngsm_Fahrt : Bool;   // langsam Fahren
      WT_nok : Bool;   // Behandlungsfehler
      WT_151 : Bool;
      WT_161 : Bool;
      res226 : Bool;
      res227 : Bool;
      Alt_Befx : USInt;   // Befehlsindex in letzter Automatikposition
      Alt_Bereichstakte : USInt;   // Bereichstakte der letzten Automatikposition
      Alt_TW_Pos : USInt;
      Alt_Verweil : DInt;   // Verweilzeit der letzten Automatikposition
      Fertigzeitpunkt : DInt;   // Systemzeit PC, wann WT voraussichtlich fertig
      Meld_Pos : USInt;   // gemerkte Kollisionposition
      WT_Typ : Byte;   // Warenträgertyp (für die Zuordnung bestimmter Ware)
      End_Ziel_Pos : USInt;   // Zielposition an die der WT
      End_Ziel_QT_Pos : USInt;   // Position die ein verwendeter QT anfahren muß
      KorrPend : Real;   // Korrekturfaktor Pendelzeit
      KorrATZ : Real;   // Korrekturfaktor Abtropfzeit
      P_PNTER : Int;   // Parameter-Pointer
      B_PNTER : Int;   // Befehls-pointer
      SaveExpo : DInt;   // gerettete Expozeit bei Zwangsräumung
      Bereichstakte : USInt;   // Takt die der WT noch im aktuellen Behandlungsbereich verbringen muß
      Variante1 : Byte;
      Variante2 : Byte;
      Variante3 : Byte;
      Variante4 : Byte;
      Variante5 : Byte;
      akt_Ziel : Int;   // aktuelles Ziel aus FB9(FC120)
      akt_CMD : Byte;   // aktueller Befehl
      WT_Kennung : Byte;   // farbliche Markierung für PC
      Speed_Up : Int;
      Speed_Dn : Int;
      Speed_Fahrt : Int;
      resI : Int;
      Aufgabezeitpunkt : DInt;   // Systemzeit PC, wann WT aufgegeben wurde
      RestTakte : Int;   // Resttakte durch die Anlage
      "Name" : String[100];
      Befehl : Array[1..20] of Struct   // * Feldlänge anpassen DB45 beachten!!
         Kennung : Byte;   // Befehlskennung
         Startpos : Byte;   // Position
         Laenge : Byte;   // Länge
         Startpos2 : Byte;
         Laenge2 : Byte;
         Sonderparam : Byte;
         Param_Ptr : Int;   // Pointer für Parameter
      END_STRUCT;
      Param_Bereich : Array[1..100] of Byte;   // * Feldlänge anpassen DB45 beachten!!
   END_VAR
BEGIN
END_DATA_BLOCK

ORGANIZATION_BLOCK "Main"   // OB1, STL, ProgramCycle
TITLE = Zyklus
{ S7_Optimized_Access := 'FALSE' }
AUTHOR : MS
// stored: AutoNumber false
   VAR_TEMP
      OB1_EV_CLASS : Byte;   // Bits 0-3 = 1 (Coming event), Bits 4-7 = 1 (Event class 1)
      OB1_SCAN_1 : Byte;   // 1 (Cold restart scan 1 of OB 1), 3 (Scan 2-n of OB 1)
      OB1_PRIORITY : Byte;   // 1 (Priority of 1 is lowest)
      OB1_OB_NUMBR : Byte;   // 1 (Organization block 1, OB1)
      OB1_RESERVED_1 : Byte;   // Reserved for system
      OB1_RESERVED_2 : Byte;   // Reserved for system
      OB1_PREV_CYCLE : Int;   // Cycle time of previous OB1 scan (milliseconds)
      OB1_MIN_CYCLE : Int;   // Minimum cycle time of OB1 (milliseconds)
      OB1_MAX_CYCLE : Int;   // Maximum cycle time of OB1 (milliseconds)
      OB1_DATE_TIME : Date_And_Time;   // Date and time OB1 started
   END_VAR
BEGIN

NETWORK
TITLE = 
//-------------------------
//Zykluszeit merken
//-------------------------
      L     #OB1_PREV_CYCLE;
      T     "DI_FW_MANAGER".akt_CT;
      L     "DI_FW_MANAGER".max_CT;
      <I;
      JC    writ;
      L     "DI_FW_MANAGER".akt_CT;
writ: T     "DI_FW_MANAGER".max_CT;
//-------------------------
//neue Anlagenkonfiguration
//-------------------------
      AN    "DB_ANLAGE".BA.newConfig;
      JC    nCfg;
      CALL  "FC_newConfig"
      ( Anlauf := FALSE
      );
nCfg: NOP   0;

//------------------------------
//Flankenauswertung Taktmerker
//------------------------------
      CALL  "Taktmerker";
//-------------------------
//Wochenschaltuhr
//-------------------------
      CALL  "Schaltuhr";
      CALL  "Uhrzeit_WSU", "Uhrzeit";

//------------------------------
//Zeiten aktualisieren
//------------------------------
      A     "Imp_1Hz";
      CC    "FC_EXPO_TIME";
//-------------------------
//PNOZ-Kommunikation
//-------------------------
      CALL  "Komm_PNOZ";
//-------------------------
//Eingänge/Eingaben lesen
//-------------------------
      CALL  "FC_DP_Error";
      CALL  "FU_Read";
      CALL  "FC_INPUT";
      CALL  "FC_SIMULATION";
//-------------------------
//Analogwerterfassung
//-------------------------
      CALL  "Analogeingabe";
//-------------------------
//Betriebsarten setzen
//-------------------------
      CALL  "BA_WXL";
//-------------------------
//Optimierung
//-------------------------
      CALL  "FC_Optimierung";
//-------------------------
//WT-Verwaltung
//-------------------------
      CALL  "FC_WT_MANAGER";
//-------------------------
//Fahrwagenverwaltung
//-------------------------
      CALL  "FC_Hilfsfuntionen";
//----------------------------------
//Pos-Reservierung überarbeiten
//----------------------------------
      CALL  "FC_FW_RES_QZ";
//----------------------------------
// FW-Verwaltung (nur bei Auftrag)
//----------------------------------
      CALL  "FB_FW_Auftrag", "DI_FW_Auftrag_DB";
//-------------------------
//Fahrwagen bearbeiten
//-------------------------
      CALL  "FB_FW_MANAGER", "DI_FW_MANAGER"
      ( CallDBNr := 
      );
//-------------------------
//Badverwaltung
//-------------------------
      CALL  "FC_Pos_Manager";
//-------------------------
//Ladungszähler
//-------------------------
      CALL  "FC_Zaehler";
      CALL  "FC_DoPu";
//-------------------------
//Anlagenfunktionen
//-------------------------
      CALL  "Peripherie";
      CALL  "FC_Niveau_St";
//-------------------------
//Alarmbehandlung gesamt
//-------------------------
      CALL  "Alarme";

//-------------------------
//Ausgänge schreiben
//-------------------------
      CALL  "FC_OUTPUT";
      CALL  "FU_Write";
//-------------------------
//Daten bereitstellen
//-------------------------
      CALL  "FC_Copy_Daten_Heraeus";

      BE;
END_ORGANIZATION_BLOCK

FUNCTION "FC_newConfig" : Void   // FC49, STL
{ S7_Optimized_Access := 'FALSE' }
AUTHOR : MS
// stored: AutoNumber false
   VAR_INPUT
      Anlauf : Bool;   // SPS befindet sich im Anlauf von Stop-->Run
   END_VAR
   VAR_TEMP
      DB_length : UDInt;
      DB_Nr_1 : DB_ANY;
      I_Max : Real;
      U_Max : Real;
      HW_Ink : DInt;
      akt_Adr : DWord;
      old_Adr : DWord;
      T_Nr : Int;
      RetValue : Int;
      DB_Nr : Word;
      RetLeng : Word;
      DB_Kette : Word;
      attrib : Byte;
      count : Byte;
      HW_count : Byte;
      minPos : Byte;
      maxPos : Byte;
      RefPos : Byte;
      Abstand : Byte;
      PosR1 : Byte;
      PosR2 : Byte;
      PosR3 : Byte;
      PosR4 : Byte;
      PosR5 : Byte;
      AnzFW : Byte;
      Absli1 : Byte;
      Absli2 : Byte;
      Absli3 : Byte;
      Absli4 : Byte;
      Absli5 : Byte;
      Absre1 : Byte;
      Absre2 : Byte;
      Absre3 : Byte;
      Absre4 : Byte;
      Absre5 : Byte;
      akt_Ebene : Byte;
      new_Ebene : Byte;
      akt_Reihe : Byte;
      first_chk : Bool;
      sub : Bool;
      old : Bool;
      wrtProt : Bool;
   END_VAR
BEGIN

NETWORK
TITLE = nach SPS-Anlauf wird nur eine Messstelle pro Zyklus bearbeitet
      A     #Anlauf;
      JC    ok;

      A     "DB_ANLAGE".BA.Automat_ein;
      BEC;

      L     "DB_ANLAGE".config.ANZ_FW;
reFC: T     #count;
      L     0;
      <=I;
      JC    QTC;
      L     #count;
      +     10;
      T     #DB_Nr;

      OPN   DB [#DB_Nr];
      A     %DBX0.1;  //"DI_FW_1".ZST.AKTIV
      BEC;
      L     #count;
      LOOP  reFC;

QTC:  L     "DB_ANLAGE".config.ANZ_QT;
reQC: T     #count;
      L     0;
      <=I;
      JC    ok;
      L     #count;
      +     30;
      T     #DB_Nr;

      OPN   DB [#DB_Nr];
      A     %DBX0.1;  //"DI_QT_1".ZST.AKTIV
      BEC;
      L     #count;
      LOOP  reQC;

ok:   L     "DB_POS".POS[1].IncPos;  //Position in Inkrementen
      L     0;
      <>D;
      =     #old;

      L     "DB_ANLAGE".config.ANZ_Pos;
      T     "DB_POS".ANZAHL;

oldA: L     53;
      T     #DB_Nr_1;

      CALL  ATTR_DB
      ( REQ       := true,
        DB_NUMBER := #DB_Nr_1,
        RET_VAL   := #RetValue,
        DB_LENGTH := #DB_length,
        ATTRIB    := #attrib
      );

      L     #RetValue;  //Fehler Db nicht vorhanden usw.
      L     0;
      <>I;
      O(;
      L     #DB_length;
      L     0;  // optimierter Baustein
      ==I;
      );
      R     "DB_ANLAGE".config.HW_exist;
      JC    RDef;

      A     #wrtProt;  //DB schreibgeschützt
      JC    RDef;

      L     "DB_ANLAGE".config2.Anzahl_HW;
      T     "DB_HW".Anzahl;
      L     0;
      <>I;
      =     "DB_ANLAGE".config.HW_exist;

//Reihendefinition
RDef: L     "DB_ANLAGE".config.Reihen_Cnfg.EndePos_R1;  //Korrektur
      L     1;
      <I;
      JC    Korr;
      L     "DB_ANLAGE".config.Reihen_Cnfg.EndePos_R1;  //Korrektur
      L     "DB_ANLAGE".config.ANZ_Pos;
      >I;
      JC    Korr;
      JU    go;
Korr: L     "DB_ANLAGE".config.ANZ_Pos;
      T     "DB_ANLAGE".config.Reihen_Cnfg.EndePos_R1;  //Korrektur

go:   L     1;
      T     #akt_Reihe;

      L     32;
      SLD   3;
      T     #akt_Adr;  //Adresse Reihen_Cnfg.EndePos_Rx

      L     1;
retP: T     #count;
      L     "DB_ANLAGE".config.ANZ_Pos;
      >I;
      JC    xF;

reRC: OPN   "DB_ANLAGE";
      L     DBW [#akt_Adr];  //"DB_ANLAGE".config.Reihen_Cnfg.EndePos_R1
      L     0;  //letzte Definierte Stelle bereits geladen
      ==I;
      JC    WPOS;

      L     #count;
      L     DBW [#akt_Adr];  //"DB_ANLAGE".config.Reihen_Cnfg.EndePos_R1
      <=I;
      JC    WPOS;

      L     #akt_Reihe;  //nächste Reihe außerhalb Gültigkeit
      L     5;
      >=I;
      JC    WPOS;

      L     #akt_Reihe;  //nächste Reihe hat begonnen
      +     1;
      T     #akt_Reihe;

      L     2;  //nächste Config-Adresse laden
      SLD   3;
      L     #akt_Adr;
      +D;
      T     #akt_Adr;
      JU    reRC;

WPOS: L     #count;
      L     "DB_POS".LENG;
      *I;
      L     "DB_POS".Offset;
      +I;
      SLD   3;
      LAR1;

      OPN   "DB_POS";
      L     #akt_Reihe;
      T     DBB [AR1, P#4.0];  //"DB_POS".POS[0].Reihe

      L     0;
      T     DBB [AR1, P#18.0];  //LZ-Nr1 im Bad
      T     DBB [AR1, P#19.0];  //LZ-Nr2 im Bad

      A     #old;
      ON    "DB_ANLAGE".BA.Simulation;
      JC    NNEW;

      OPN   "DB_POS";
      L     #count;
      L     1000;
      *D;
      T     DBD [AR1, P#22.0];  //Position in Inkrementen

NNEW: A     "DB_ANLAGE".config.Pos_absolut;
      JC    Nabs;

      OPN   "DB_POS";
      L     #count;
      L     5;
      *D;
      T     DBD [AR1, P#22.0];  //Position in Inkrementen

Nabs: OPN   "DB_POS";
      L     0;
      L     DBB [AR1, P#13.0];  //Stand_Nr
      ==I;
      JC    nexP;
      DEC   1;
      L     "DB_BE_Stand".Anzahl;
      >I;
      JC    nexP;
      CAC;
      L     "DB_BE_Stand".leng;
      *D;
      L     "DB_BE_Stand".Offset;
      +D;
      SLD   3;
      LAR1;
      OPN   "DB_BE_Stand";
      L     #count;
      T     DBB [AR1, P#0.0];  //Pos_Nr im BE_DB

nexP: L     #count;
      L     1;
      +I;
      JU    retP;

xF:   L     "DB_ANLAGE".config.ANZ_FW;
retF: T     #count;
      L     0;
      <=I;
      JC    DZ;

      L     #count;
      DEC   1;
      L     10;
      *I;
      +     100;
      SLD   3;
      LAR1;

      OPN   "DB_ANLAGE";
      L     DBW [AR1, P#0.0];  //"DB_ANLAGE".FW1.FW_min
      T     #minPos;
      L     DBW [AR1, P#2.0];  //"DB_ANLAGE".FW1.FW_max
      T     #maxPos;
      L     DBW [AR1, P#4.0];  //"DB_ANLAGE".FW1.RefPos
      T     #RefPos;
      L     DBW [AR1, P#6.0];  //"DB_ANLAGE".FW1.T_Nr
      T     #T_Nr;

      L     #minPos;
      L     "DB_ANLAGE".config.Reihen_Cnfg.EndePos_R1;
      <=I;
      L     1;
      JC    RF;
      L     #minPos;
      L     "DB_ANLAGE".config.Reihen_Cnfg.EndePos_R2;
      <=I;
      L     2;
      JC    RF;
      L     #minPos;
      L     "DB_ANLAGE".config.Reihen_Cnfg.EndePos_R3;
      <=I;
      L     3;
      JC    RF;
      L     #minPos;
      L     "DB_ANLAGE".config.Reihen_Cnfg.EndePos_R4;
      <=I;
      L     4;
      JC    RF;
      L     #minPos;
      L     "DB_ANLAGE".config.Reihen_Cnfg.EndePos_R5;
      <=I;
      L     5;
      JC    RF;
      L     0;
RF:   T     #akt_Reihe;

      L     #count;
      L     10;
      +I;
      T     #DB_Nr;

      OPN   DB [#DB_Nr];
      L     %DBB2;  //Istposition
      L     0;
      <>I;
      JC    okF;

      L     #minPos;
      T     %DBB2;  //Istposition

okF:  L     #minPos;
      T     %DBB194;  //"DI_FW_1".PAR.Fahrt.FAHRBEREICH_MIN

      L     #maxPos;
      T     %DBB195;  //"DI_FW_1".PAR.Fahrt.FAHRBEREICH_MAX

      L     #RefPos;
      T     %DBB196;  //"DI_FW_1".PAR.Fahrt.REF_Pos

      L     #T_Nr;
      T     %DBW184;  //"DI_FW_1".PAR.TIMER_NR

      L     #count;
      T     %DBB182;  //"DI_FW_1".PAR.FW_Nr

      L     #akt_Reihe;
      T     %DBB186;  //"DI_FW_1".PAR.Reihe

      SET;
      =     %DBX0.2;  //"DI_FW_1".ZST.FEHLER
      =     %DBX53.4;  //"DI_FW_1".IN.Com_Reset

      L     #count;
      DEC   1;
      JU    retF;

DZ:   L     0;
      L     "DB_ANLAGE".config.Anz_DZ;
      ==I;
      JC    DP;
      T     "DB_Zaehler".Anz_Beck;

DP:   L     0;
      L     "DB_ANLAGE".config.Anz_DP;
      ==I;
      JC    nxt;
      T     "DB_DP".Anz_DP;
      T     "DB_Panel_DP".Anz_DP;

nxt:  SET;
      R     "DB_ANLAGE".BA.newConfig;

END_FUNCTION

FUNCTION "Taktmerker" : Void
{ S7_Optimized_Access := 'TRUE' }
VERSION : 0.1

BEGIN
	(* Systemtakt (MB50 Clock_Byte) 
	auf positive Flanke (Impuls) in MB52
	Altmerkerbyte MB51 *)
	
	"MB_Imp_ClockByte" := ("Clock_Byte" XOR "MB_SystemAltTakt") AND "Clock_Byte";
	"MB_SystemAltTakt" := "Clock_Byte";
END_FUNCTION

FUNCTION "Schaltuhr" : Void
{ S7_Optimized_Access := 'TRUE' }
VERSION : 0.1
   VAR_TEMP 
      return : Int;
      i : Int;
      j : Int;
      Minuten : Array[0..30] of Struct   // Array mit die Minuten von Sonntag 00:00 (Ein- und Ausschaltung)
         Min : DInt;
      END_STRUCT;
      Start_Aus : Bool;
      Switch_1 : Byte;   // Kann ein- oder ausschalten, es häng von Start_Aus ab
      Switch_2 : Byte;
   END_VAR


BEGIN
	//------------------
	//Uhrzeit stellen
	//------------------
	//SPS Zeit holen nach Tastendruck
	IF "DB_Schaltuhr".SPS_Zeit_holen THEN
	    "DB_Schaltuhr".Date_Time_Visu := "Uhrzeit".aktDatum;
	    "DB_Schaltuhr".SPS_Zeit_holen := FALSE;
	END_IF;
	
	//SPS Zeit stellen nach Tastendruck
	IF "DB_Schaltuhr".SPS_Zeit_Stellen THEN
	    #return := WR_LOC_T(LOCTIME := "DB_Schaltuhr".Date_Time_Visu,DST := FALSE);
	    "DB_Schaltuhr".SPS_Zeit_Stellen := FALSE;
	END_IF;
	
	//-------------------------
	//Betriebsart aus Visu
	//-------------------------
	CASE "DB_Schaltuhr".BA_Visu OF
	    0:  //Aus
	        "Uhrzeit".BA_Uhr_Ein := FALSE;
	        "Uhrzeit".BA_Uhr_Dauer := FALSE;
	    1:  // Dauerbetrieb
	        "Uhrzeit".BA_Uhr_Ein := FALSE;
	        "Uhrzeit".BA_Uhr_Dauer := TRUE;
	    2:  // Ein
	        "Uhrzeit".BA_Uhr_Ein := TRUE;
	        "Uhrzeit".BA_Uhr_Dauer := FALSE;
	END_CASE;
	
	//-------------------------
	//Arbeitszeiten Übernehmen
	//-------------------------
	IF "DB_Schaltuhr".Taste_uebernehmen THEN
	    
	    "Schaltuhr_Pruefung"(Uebernehmen := "DB_Schaltuhr".Taste_uebernehmen,
	                            Array => #Minuten,
	                            Error => "DB_Schaltuhr".nichtOK,
	                            Start_Aus => #Start_Aus);
	    
	    "DB_Schaltuhr".Taste_uebernehmen := FALSE;
	    
	    IF "DB_Schaltuhr".nichtOK THEN
	        RETURN; //Ende wenn fehlerhafte Einträge
	    END_IF;
	    
	    "DB_Schaltuhr".Uebernommen := TRUE;
	    
	    IF #Start_Aus THEN
	        #Switch_1 := 2;
	        #Switch_2 := 1;
	    ELSE
	        #Switch_1 := 1;
	        #Switch_2 := 2;
	    END_IF;
	    
	    // Array transferieren. -1 ist der Ende des Arrays
	    FOR #i := 0 TO 27 DO
	        #j := #i;
	        
	        IF #Minuten[#i].Min = dint#-1 THEN
	            EXIT;
	        END_IF;
	        
	        "Uhrzeit".ProfileWeek[#i].MinWeek := DINT_TO_INT(#Minuten[#i].Min);
	        
	        IF #i MOD 2 = 0 THEN
	            "Uhrzeit".ProfileWeek[#i].State := #Switch_1;
	        ELSE
	            "Uhrzeit".ProfileWeek[#i].State := #Switch_2;
	        END_IF;
	        
	    END_FOR;
	    
	    //Restliche Struktur löschen
	    FOR #i := #j TO 27 DO
	        "Uhrzeit".ProfileWeek[#i].MinWeek := 0;
	        "Uhrzeit".ProfileWeek[#i].State := 0;
	    END_FOR;
	    
	END_IF;
	
END_FUNCTION

FUNCTION "Schaltuhr_Pruefung" : Void
{ S7_Optimized_Access := 'TRUE' }
VERSION : 0.1
   VAR_INPUT 
      Uebernehmen : Bool;
   END_VAR

   VAR_OUTPUT 
      "Array" : Array[0..30] of Struct   // Array mit die Minuten von Sonntag 00:00 (Ein- und Ausschaltung)
         Min : DInt;
      END_STRUCT;
      Error : Bool;
      Start_Aus : Bool;   // =1 heißt dass der erste State eine Ausschaltung ist
   END_VAR

   VAR_TEMP 
      i : Int;
      j : Int;
      pruef : Int;
      anfang : Int;
   END_VAR


BEGIN
	
	IF #Uebernehmen = true THEN
	    
	    #j := 0; // Wochenschaltpunkte.
	    #pruef := 0; //Prüfparameter, muss immer 0 oder 1 sein, 0 am Ende.
	    #anfang := 0;//Anfangsparameter: -1 heißt mit Ausschaltung anfangen, 1 heißt mit Einschaltung anfangen
	    #Start_Aus := false;
	    #Error := false;
	    FILL_BLK(IN:=dint#0,
	             COUNT:=31,
	             OUT=>#Array[0].Min);
	    
	FOR #i := 1 TO 7 DO //Sonntag bis Samstag
	    
	//--------------------------
	//1te Spur am Tag
	//--------------------------
	  //Begin ---------------------------------------------------------------------------------------
	  IF "DB_Schaltuhr".Tag_aktiv[#i].AZ_Begin1_aktiv=true THEN //Wenn Zeit aktiv
	    
	    #Array[#j].Min := TOD_TO_DINT(DTL_TO_TOD("DB_Schaltuhr".Tag[#i].AZ_Begin1))/60000+(#i-1)*1440; //Kopiere im Array
	    #j := #j+1; //Array+1
	    #pruef := #pruef + 1;
	    
	    IF #anfang = 0 THEN 
	      #anfang := 1;
	    END_IF;
	    
	    IF #pruef <> 1 THEN
	      #Error := true;
	    END_IF;
	    
	  END_IF;
	  //Ende ------------------------------------------------------------------------------------------
	  
	  //Begin ---------------------------------------------------------------------------------------
	  IF "DB_Schaltuhr".Tag_aktiv[#i].AZ_Ende1_aktiv=true THEN//Wenn Zeit aktiv
	    
	      #Array[#j].Min := TOD_TO_DINT(DTL_TO_TOD("DB_Schaltuhr".Tag[#i].AZ_Ende1))/60000+(#i-1)*1440;//Kopiere im Array
	   #j := #j+1;//Array+1
	   #pruef := #pruef - 1;
	   
	   IF #anfang = 0 THEN
	     #anfang := -1;
	     #pruef := 0; //Pruefparameter wieder auf Null
	   END_IF;
	    
	   IF #pruef <> 0 THEN
	      #Error := true;
	   END_IF;
	    
	  END_IF;
	  //Ende ------------------------------------------------------------------------------------------
	  
